// Action: select text with ID 19: go back;
	L 	19;
	T 	button_1_text;

//---------------------------------
// --- TRANSITION TO S480 ---
//---------------------------------

// Transition Logic
	SET;	// make sure RLO is high so the transition can happen when no conditions present

	A	button_1_pushed; 	// button “go back
	JCN L35;

	L   480;
	T   stepnumber;

L35: NOP 0;


//---------------------------------
// Actions (last scan)
// This is immediately executed once the stepnumber changes
//---------------------------------
	L	stepnumber;
	L	previous_stepnumber;
	<>I;
	JCN D35;

// Action: hide button_1
	CLR;
	=	button_1_visible;


D35: NOP 0;

//---------------------------------
// End of network: jump here if step not active
// Jump to end of this FB if the step has been active to avoid
// execution of another step in the same scan
//---------------------------------
	JU	ENDS;
J35: NOP 0;

//__phase_example_Step_470_END

NETWORK
TITLE = Step 480
//___phase_example_Step_480_
//================================
// test 3 buttons
//================================

// skip this network if stepnumber not equal to 480
	L 	stepnumber;
	L 	480;
	==I;
	JCN J36;

//---------------------------------
// Actions (continuouss)
//---------------------------------

// Action: show button_1
	SET;
	=	button_1_visible;

// Action: select text with ID 16: continue;
	L 	16;
	T 	button_1_text;

// Action: show button_2
	SET;
	=	button_2_visible;

// Action: select text with ID 18: cancel;
	L 	18;
	T 	button_2_text;

// Action: show button_3
	SET;
	=	button_3_visible;

// Action: select text with ID 19: go back;
	L 	19;
	T 	button_3_text;

//---------------------------------
// --- TRANSITION TO S490 ---
//---------------------------------

// Transition Logic
	SET;	// make sure RLO is high so the transition can happen when no conditions present

	A	button_1_pushed; 	// button “continue”
	A	button_2_pushed; 	// button “cancel”
	A	button_3_pushed; 	// button “go back”
	JCN L36;

	L   490;
	T   stepnumber;

L36: NOP 0;


//---------------------------------
// Actions (last scan)
// This is immediately executed once the stepnumber changes
//---------------------------------
	L	stepnumber;
	L	previous_stepnumber;
	<>I;
	JCN D36;

// Action: hide button_1
	CLR;
	=	button_1_visible;

// Action: hide button_2
	CLR;
	=	button_2_visible;

// Action: hide button_3
	CLR;
	=	button_3_visible;


D36: NOP 0;

//---------------------------------
// End of network: jump here if step not active
// Jump to end of this FB if the step has been active to avoid
// execution of another step in the same scan
//---------------------------------
	JU	ENDS;
J36: NOP 0;

//__phase_example_Step_480_END

NETWORK
TITLE = Step 490
//___phase_example_Step_490_
//================================
// test 4 buttons => not foreseen in the template, so should log an error
//================================

// skip this network if stepnumber not equal to 490
	L 	stepnumber;
	L 	490;
	==I;
	JCN J37;

//---------------------------------
// Actions (continuouss)
//---------------------------------

// Action: show button_1
	SET;
	=	button_1_visible;

// Action: select text with ID 16: continue;
	L 	16;
	T 	button_1_text;

// Action: show button_2
	SET;
	=	button_2_visible;

// Action: select text with ID 18: cancel;
	L 	18;
	T 	button_2_text;

// Action: show button_3
	SET;
	=	button_3_visible;

// Action: select text with ID 19: go back;
	L 	19;
	T 	button_3_text;

//---------------------------------
// --- TRANSITION TO S510 ---
//---------------------------------

// Transition Logic
	SET;	// make sure RLO is high so the transition can happen when no conditions present

	A	button_1_pushed; 	// button “continue”
	A	button_2_pushed; 	// button “cancel”
	A	button_3_pushed; 	// button “go back”
	JCN L37;

	L   510;
	T   stepnumber;

L37: NOP 0;


//---------------------------------
// Actions (last scan)
// This is immediately executed once the stepnumber changes
//---------------------------------
	L	stepnumber;
	L	previous_stepnumber;
	<>I;
	JCN D37;

// Action: hide button_1
	CLR;
	=	button_1_visible;

// Action: hide button_2
	CLR;
	=	button_2_visible;

// Action: hide button_3
	CLR;
	=	button_3_visible;


D37: NOP 0;

//---------------------------------
// End of network: jump here if step not active
// Jump to end of this FB if the step has been active to avoid
// execution of another step in the same scan
//---------------------------------
	JU	ENDS;
J37: NOP 0;

//__phase_example_Step_490_END

NETWORK
TITLE = Step 510
//___phase_example_Step_510_
//================================
// test message
//================================

// skip this network if stepnumber not equal to 510
	L 	stepnumber;
	L 	510;
	==I;
	JCN J38;

//---------------------------------
// Actions (continuouss)
//---------------------------------

// Action: message “add the manual ingredients”;
	L 	21;
	T 	message;

//---------------------------------
// --- TRANSITION TO S520 ---
//---------------------------------

// Transition Logic
	SET;	// make sure RLO is high so the transition can happen when no conditions present

	JCN L38;

	L   520;
	T   stepnumber;

L38: NOP 0;


//---------------------------------
// Actions (last scan)
// This is immediately executed once the stepnumber changes
//---------------------------------
	L	stepnumber;
	L	previous_stepnumber;
	<>I;
	JCN D38;

// Action: clear message;
	L 	0;
	T 	message;


D38: NOP 0;

//---------------------------------
// End of network: jump here if step not active
// Jump to end of this FB if the step has been active to avoid
// execution of another step in the same scan
//---------------------------------
	JU	ENDS;
J38: NOP 0;

//__phase_example_Step_510_END

NETWORK
TITLE = Step 520
//___phase_example_Step_520_
//================================
// test falseword with two words in transition
//================================

// skip this network if stepnumber not equal to 520
	L 	stepnumber;
	L 	520;
	==I;
	JCN J39;

//---------------------------------
// Actions (continuouss)
//---------------------------------

//---------------------------------
// --- TRANSITION TO S530 ---
//---------------------------------

// Transition Logic
	SET;	// make sure RLO is high so the transition can happen when no conditions present

	AN	XV003_OPN; 	// XV003 not opened
	JCN L39;

	L   530;
	T   stepnumber;

L39: NOP 0;


D39: NOP 0;

//---------------------------------
// End of network: jump here if step not active
// Jump to end of this FB if the step has been active to avoid
// execution of another step in the same scan
//---------------------------------
	JU	ENDS;
J39: NOP 0;

//__phase_example_Step_520_END

NETWORK
TITLE = Step 530
//___phase_example_Step_530_
//================================
// test trueword with multiple words in action
//================================

// skip this network if stepnumber not equal to 530
	L 	stepnumber;
	L 	530;
	==I;
	JCN J40;

//---------------------------------
// Actions (continuouss)
//---------------------------------

// Action: move to open position XV003
	SET;
	=	XV003_CMD;

//---------------------------------
// --- TRANSITION TO S540 ---
//---------------------------------

// Transition Logic
	SET;	// make sure RLO is high so the transition can happen when no conditions present

	JCN L40;

	L   540;
	T   stepnumber;

L40: NOP 0;


D40: NOP 0;

//---------------------------------
// End of network: jump here if step not active
// Jump to end of this FB if the step has been active to avoid
// execution of another step in the same scan
//---------------------------------
	JU	ENDS;
J40: NOP 0;

//__phase_example_Step_530_END

NETWORK
TITLE = Step 540
//___phase_example_Step_540_
//================================
// test putting controller in auto with pulseword
//================================

// skip this network if stepnumber not equal to 540
	L 	stepnumber;
	L 	540;
	==I;
	JCN J41;

//---------------------------------
// Actions (continuouss)
//---------------------------------

// Action: FIC001 auto
	SET;
	=	FIC001_AUT;

//---------------------------------
// --- TRANSITION TO S550 ---
//---------------------------------

// Transition Logic
	SET;	// make sure RLO is high so the transition can happen when no conditions present

	JCN L41;

	L   550;
	T   stepnumber;

L41: NOP 0;


D41: NOP 0;

//---------------------------------
// End of network: jump here if step not active
// Jump to end of this FB if the step has been active to avoid
// execution of another step in the same scan
//---------------------------------
	JU	ENDS;
J41: NOP 0;

//__phase_example_Step_540_END

NETWORK
TITLE = Step 550
//___phase_example_Step_550_
//================================
// test putting controller in auto with pulseword consisting of multiple words
//================================

// skip this network if stepnumber not equal to 550
	L 	stepnumber;
	L 	550;
	==I;
	JCN J42;

//---------------------------------
// Actions (continuouss)
//---------------------------------

// Action: FIC001 switch to auto
	SET;
	=	FIC001_AUT;

//---------------------------------
// --- TRANSITION TO S560 ---
//---------------------------------

// Transition Logic
	SET;	// make sure RLO is high so the transition can happen when no conditions present

	JCN L42;

	L   560;
	T   stepnumber;

L42: NOP 0;


D42: NOP 0;

//---------------------------------
// End of network: jump here if step not active
// Jump to end of this FB if the step has been active to avoid
// execution of another step in the same scan
//---------------------------------
	JU	ENDS;
J42: NOP 0;

//__phase_example_Step_550_END

NETWORK
TITLE = Step 560
//___phase_example_Step_560_
//================================
// test with pulseword in front
//================================

// skip this network if stepnumber not equal to 560
	L 	stepnumber;
	L 	560;
	==I;
	JCN J43;

//---------------------------------
// Actions (continuouss)
//---------------------------------

// Action: auto FIC001
	SET;
	=	FIC001_AUT;

//---------------------------------
// --- TRANSITION TO S570 ---
//---------------------------------

// Transition Logic
	SET;	// make sure RLO is high so the transition can happen when no conditions present

	JCN L43;

	L   570;
	T   stepnumber;

L43: NOP 0;


D43: NOP 0;

//---------------------------------
// End of network: jump here if step not active
// Jump to end of this FB if the step has been active to avoid
// execution of another step in the same scan
//---------------------------------
	JU	ENDS;
J43: NOP 0;

//__phase_example_Step_560_END

NETWORK
TITLE = Step 570
//___phase_example_Step_570_
//================================
// test with pulseword in front
//================================

// skip this network if stepnumber not equal to 570
	L 	stepnumber;
	L 	570;
	==I;
	JCN J44;

//---------------------------------
// Actions (continuouss)
//---------------------------------

// Action: switch to auto FIC001
	SET;
	=	FIC001_AUT;

//---------------------------------
// --- TRANSITION TO S580 ---
//---------------------------------

// Transition Logic
	SET;	// make sure RLO is high so the transition can happen when no conditions present

	JCN L44;

	L   580;
	T   stepnumber;

L44: NOP 0;


D44: NOP 0;

//---------------------------------
// End of network: jump here if step not active
// Jump to end of this FB if the step has been active to avoid
// execution of another step in the same scan
//---------------------------------
	JU	ENDS;
J44: NOP 0;

//__phase_example_Step_570_END

NETWORK
TITLE = Step 580
//___phase_example_Step_580_
//================================
// test steptime in s
//================================

// skip this network if stepnumber not equal to 580
	L 	stepnumber;
	L 	580;
	==I;
	JCN J45;

//---------------------------------
// Actions (continuouss)
//---------------------------------

//---------------------------------
// --- TRANSITION TO S590 ---
//---------------------------------

// Calculation:
	L 	steptime_s;
	L 	2.0;
	>R;
	=	B5;

// Transition Logic
	SET;	// make sure RLO is high so the transition can happen when no conditions present

	A	B5; 	// steptime > 2.0s
	JCN L45;

	L   590;
	T   stepnumber;

L45: NOP 0;


D45: NOP 0;

//---------------------------------
// End of network: jump here if step not active
// Jump to end of this FB if the step has been active to avoid
// execution of another step in the same scan
//---------------------------------
	JU	ENDS;
J45: NOP 0;

//__phase_example_Step_580_END

NETWORK
TITLE = Step 590
//___phase_example_Step_590_
//================================
// test steptime in m
//================================

// skip this network if stepnumber not equal to 590
	L 	stepnumber;
	L 	590;
	==I;
	JCN J46;

//---------------------------------
// Actions (continuouss)
//---------------------------------

//---------------------------------
// --- TRANSITION TO S600 ---
//---------------------------------

// Calculation:
	L 	steptime_m;
	L 	1.50;
	>R;
	=	B6;

// Transition Logic
	SET;	// make sure RLO is high so the transition can happen when no conditions present

	A	B6; 	// steptime > 1.50m
	JCN L46;

	L   600;
	T   stepnumber;

L46: NOP 0;


D46: NOP 0;

//---------------------------------
// End of network: jump here if step not active
// Jump to end of this FB if the step has been active to avoid
// execution of another step in the same scan
//---------------------------------
	JU	ENDS;
J46: NOP 0;

//__phase_example_Step_590_END

NETWORK
TITLE = Step 600
//___phase_example_Step_600_
//================================
// test steptime in h
//================================

// skip this network if stepnumber not equal to 600
	L 	stepnumber;
	L 	600;
	==I;
	JCN J47;

//---------------------------------
// Actions (continuouss)
//---------------------------------

//---------------------------------
// --- TRANSITION TO S610 ---
//---------------------------------

// Calculation:
	L 	steptime_h;
	L 	4.3;
	>R;
	=	B7;

// Transition Logic
	SET;	// make sure RLO is high so the transition can happen when no conditions present

	A	B7; 	// steptime > 4.3h
	JCN L47;

	L   610;
	T   stepnumber;

L47: NOP 0;


D47: NOP 0;

//---------------------------------
// End of network: jump here if step not active
// Jump to end of this FB if the step has been active to avoid
// execution of another step in the same scan
//---------------------------------
	JU	ENDS;
J47: NOP 0;

//__phase_example_Step_600_END

NETWORK
TITLE = Step 610
//___phase_example_Step_610_
//================================
// test steptime with unit separated by space => still works (because it takes the last character)
//================================

// skip this network if stepnumber not equal to 610
	L 	stepnumber;
	L 	610;
	==I;
	JCN J48;

//---------------------------------
// Actions (continuouss)
//---------------------------------

//---------------------------------
// --- TRANSITION TO S640 ---
//---------------------------------

// Calculation:
	L 	steptime_m;
	L 	1.50;
	>R;
	=	B8;

// Transition Logic
	SET;	// make sure RLO is high so the transition can happen when no conditions present

	A	B8; 	// steptime > 1.50 m
	JCN L48;

	L   640;
	T   stepnumber;

L48: NOP 0;


D48: NOP 0;

//---------------------------------
// End of network: jump here if step not active
// Jump to end of this FB if the step has been active to avoid
// execution of another step in the same scan
//---------------------------------
	JU	ENDS;
J48: NOP 0;

//__phase_example_Step_610_END

NETWORK
TITLE = Step 640
//___phase_example_Step_640_
//================================
// test steptime with variable with unit
//================================

// skip this network if stepnumber not equal to 640
	L 	stepnumber;
	L 	640;
	==I;
	JCN J49;

//---------------------------------
// Actions (continuouss)
//---------------------------------

//---------------------------------
// --- TRANSITION TO S650 ---
//---------------------------------

// Calculation:
	L 	steptime_h;
	L 	timesetting;
	>R;
	=	B9;

// Transition Logic
	SET;	// make sure RLO is high so the transition can happen when no conditions present

	A	B9; 	// steptime > timesetting
	JCN L49;

	L   650;
	T   stepnumber;

L49: NOP 0;


D49: NOP 0;

//---------------------------------
// End of network: jump here if step not active
// Jump to end of this FB if the step has been active to avoid
// execution of another step in the same scan
//---------------------------------
	JU	ENDS;
J49: NOP 0;

//__phase_example_Step_640_END

NETWORK
TITLE = Step 650
//___phase_example_Step_650_
//================================
// reset a timer
//================================

// skip this network if stepnumber not equal to 650
	L 	stepnumber;
	L 	650;
	==I;
	JCN J50;

//---------------------------------
// Actions (continuouss)
//---------------------------------

// Action: reset timer_dosing;
	L 	0.0;
	T 	timer_dosing_s;

//---------------------------------
// --- TRANSITION TO S660 ---
//---------------------------------

// Transition Logic
	SET;	// make sure RLO is high so the transition can happen when no conditions present

	JCN L50;

	L   660;
	T   stepnumber;

L50: NOP 0;


D50: NOP 0;

//---------------------------------
// End of network: jump here if step not active
// Jump to end of this FB if the step has been active to avoid
// execution of another step in the same scan
//---------------------------------
	JU	ENDS;
J50: NOP 0;

//__phase_example_Step_650_END

NETWORK
TITLE = Step 660
//___phase_example_Step_660_
//================================
// start a timer
//================================

// skip this network if stepnumber not equal to 660
	L 	stepnumber;
	L 	660;
	==I;
	JCN J51;

//---------------------------------
// Actions (continuouss)
//---------------------------------

// Action: start timer_mixing
	CLR;
	=	timer_mixing_pause;

//---------------------------------
// --- TRANSITION TO S670 ---
//---------------------------------

// Transition Logic
	SET;	// make sure RLO is high so the transition can happen when no conditions present

	JCN L51;

	L   670;
	T   stepnumber;

L51: NOP 0;


D51: NOP 0;

//---------------------------------
// End of network: jump here if step not active
// Jump to end of this FB if the step has been active to avoid
// execution of another step in the same scan
//---------------------------------
	JU	ENDS;
J51: NOP 0;

//__phase_example_Step_660_END

NETWORK
TITLE = Step 670
//___phase_example_Step_670_
//================================
// pause a timer
//================================

// skip this network if stepnumber not equal to 670
	L 	stepnumber;
	L 	670;
	==I;
	JCN J52;

//---------------------------------
// Actions (continuouss)
//---------------------------------

// Action: pause timer_circulation
	SET;
	=	timer_circulation_pause;

//---------------------------------
// --- TRANSITION TO S680 ---
//---------------------------------

// Transition Logic
	SET;	// make sure RLO is high so the transition can happen when no conditions present

	JCN L52;

	L   680;
	T   stepnumber;

L52: NOP 0;


D52: NOP 0;

//---------------------------------
// End of network: jump here if step not active
// Jump to end of this FB if the step has been active to avoid
// execution of another step in the same scan
//---------------------------------
	JU	ENDS;
J52: NOP 0;

//__phase_example_Step_670_END

NETWORK
TITLE = Step 680
//___phase_example_Step_680_
//================================
// test timer in m
//================================

// skip this network if stepnumber not equal to 680
	L 	stepnumber;
	L 	680;
	==I;
	JCN J53;

//---------------------------------
// Actions (continuouss)
//---------------------------------

//---------------------------------
// --- TRANSITION TO S690 ---
//---------------------------------

// Calculation:
	L 	timer_dosing_m;
	L 	5.2;
	>=R;
	=	B10;

// Transition Logic
	SET;	// make sure RLO is high so the transition can happen when no conditions present

	A	B10; 	// timer_dosing >= 5.2 m
	JCN L53;

	L   690;
	T   stepnumber;

L53: NOP 0;


D53: NOP 0;

//---------------------------------
// End of network: jump here if step not active
// Jump to end of this FB if the step has been active to avoid
// execution of another step in the same scan
//---------------------------------
	JU	ENDS;
J53: NOP 0;

//__phase_example_Step_680_END

NETWORK
TITLE = Step 690
//___phase_example_Step_690_
//================================
// test timer with variable with unit
//================================

// skip this network if stepnumber not equal to 690
	L 	stepnumber;
	L 	690;
	==I;
	JCN J54;

//---------------------------------
// Actions (continuouss)
//---------------------------------

//---------------------------------
// --- TRANSITION TO S700 ---
//---------------------------------

// Calculation:
	L 	timer_circulation_h;
	L 	timesetting;
	<R;
	=	B11;

// Transition Logic
	SET;	// make sure RLO is high so the transition can happen when no conditions present

	A	B11; 	// timer_circulation < timesetting
	JCN L54;

	L   700;
	T   stepnumber;

L54: NOP 0;


D54: NOP 0;

//---------------------------------
// End of network: jump here if step not active
// Jump to end of this FB if the step has been active to avoid
// execution of another step in the same scan
//---------------------------------
	JU	ENDS;
J54: NOP 0;

//__phase_example_Step_690_END

NETWORK
TITLE = Step 700
//___phase_example_Step_700_
//================================
// test putting a controller in manual
//================================

// skip this network if stepnumber not equal to 700
	L 	stepnumber;
	L 	700;
	==I;
	JCN J55;

//---------------------------------
// Actions (continuouss)
//---------------------------------

// Action: FIC001 manual
	CLR;
	=	FIC001_AUT;

//---------------------------------
// --- TRANSITION TO S710 ---
//---------------------------------

// Transition Logic
	SET;	// make sure RLO is high so the transition can happen when no conditions present

	JCN L55;

	L   710;
	T   stepnumber;

L55: NOP 0;


D55: NOP 0;

//---------------------------------
// End of network: jump here if step not active
// Jump to end of this FB if the step has been active to avoid
// execution of another step in the same scan
//---------------------------------
	JU	ENDS;
J55: NOP 0;

//__phase_example_Step_700_END

NETWORK
TITLE = Step 710
//___phase_example_Step_710_
//================================
// test putting a controller in manual while changing the output value
//================================

// skip this network if stepnumber not equal to 710
	L 	stepnumber;
	L 	710;
	==I;
	JCN J56;

//---------------------------------
// Actions (first scan)
//---------------------------------
	A	initial_scan;
	JCN   C56;

// Action: FIC001_VAL_OUT = 20.0;
	L 	20.0;
	T 	FIC001_VAL_OUT;

// Action: FIC001_SET_OUT = true
	SET;
	=	FIC001_SET_OUT;

	JU	D56;	//skip the continuous steps and transition during the initial scan
C56: NOP   0;


//---------------------------------
// Actions (continuouss)
//---------------------------------

// Action: FIC001 manual 20.0
	CLR;
	=	FIC001_AUT;

// Action: FIC001_SET_OUT = false
	CLR;
	=	FIC001_SET_OUT;

//---------------------------------
// --- TRANSITION TO S720 ---
//---------------------------------

// Transition Logic
	SET;	// make sure RLO is high so the transition can happen when no conditions present

	JCN L56;

	L   720;
	T   stepnumber;

L56: NOP 0;


D56: NOP 0;

//---------------------------------
// End of network: jump here if step not active
// Jump to end of this FB if the step has been active to avoid
// execution of another step in the same scan
//---------------------------------
	JU	ENDS;
J56: NOP 0;

//__phase_example_Step_710_END

NETWORK
TITLE = Step 720
//___phase_example_Step_720_
//================================
// test putting a controller in manual while changing the output value that has a unit
//================================

// skip this network if stepnumber not equal to 720
	L 	stepnumber;
	L 	720;
	==I;
	JCN J57;

//---------------------------------
// Actions (first scan)
//---------------------------------
	A	initial_scan;
	JCN   C57;

// Action: FIC001_VAL_OUT = 20.0;
	L 	20.0;
	T 	FIC001_VAL_OUT;

// Action: FIC001_SET_OUT = true
	SET;
	=	FIC001_SET_OUT;

	JU	D57;	//skip the continuous steps and transition during the initial scan
C57: NOP   0;


//---------------------------------
// Actions (continuouss)
//---------------------------------

// Action: FIC001 manual 20.0 Hz
	CLR;
	=	FIC001_AUT;

// Action: FIC001_SET_OUT = false
	CLR;
	=	FIC001_SET_OUT;

//---------------------------------
// --- TRANSITION TO S730 ---
//---------------------------------

// Transition Logic
	SET;	// make sure RLO is high so the transition can happen when no conditions present

	JCN L57;

	L   730;
	T   stepnumber;

L57: NOP 0;


D57: NOP 0;

//---------------------------------
// End of network: jump here if step not active
// Jump to end of this FB if the step has been active to avoid
// execution of another step in the same scan
//---------------------------------
	JU	ENDS;
J57: NOP 0;

//__phase_example_Step_720_END

NETWORK
TITLE = Step 730
//___phase_example_Step_730_
//================================
// without space
//================================

// skip this network if stepnumber not equal to 730
	L 	stepnumber;
	L 	730;
	==I;
	JCN J58;

//---------------------------------
// Actions (first scan)
//---------------------------------
	A	initial_scan;
	JCN   C58;

// Action: FIC001_VAL_OUT = 20.0;
	L 	20.0;
	T 	FIC001_VAL_OUT;

// Action: FIC001_SET_OUT = true
	SET;
	=	FIC001_SET_OUT;

	JU	D58;	//skip the continuous steps and transition during the initial scan
C58: NOP   0;


//---------------------------------
// Actions (continuouss)
//---------------------------------

// Action: FIC001 manual 20.0Hz
	CLR;
	=	FIC001_AUT;

// Action: FIC001_SET_OUT = false
	CLR;
	=	FIC001_SET_OUT;

//---------------------------------
// --- TRANSITION TO S740 ---
//---------------------------------

// Transition Logic
	SET;	// make sure RLO is high so the transition can happen when no conditions present

	JCN L58;

	L   740;
	T   stepnumber;

L58: NOP 0;


D58: NOP 0;

//---------------------------------
// End of network: jump here if step not active
// Jump to end of this FB if the step has been active to avoid
// execution of another step in the same scan
//---------------------------------
	JU	ENDS;
J58: NOP 0;

//__phase_example_Step_730_END

NETWORK
TITLE = Step 740
//___phase_example_Step_740_
//================================
// put PID controller in auto
//================================

// skip this network if stepnumber not equal to 740
	L 	stepnumber;
	L 	740;
	==I;
	JCN J59;

//---------------------------------
// Actions (continuouss)
//---------------------------------

// Action: FIC001 auto
	SET;
	=	FIC001_AUT;

//---------------------------------
// --- TRANSITION TO S750 ---
//---------------------------------

// Transition Logic
	SET;	// make sure RLO is high so the transition can happen when no conditions present

	JCN L59;

	L   750;
	T   stepnumber;

L59: NOP 0;


D59: NOP 0;

//---------------------------------
// End of network: jump here if step not active
// Jump to end of this FB if the step has been active to avoid
// execution of another step in the same scan
//---------------------------------
	JU	ENDS;
J59: NOP 0;

//__phase_example_Step_740_END

NETWORK
TITLE = Step 750
//___phase_example_Step_750_
//================================
// auto with setpoint
//================================

// skip this network if stepnumber not equal to 750
	L 	stepnumber;
	L 	750;
	==I;
	JCN J60;

//---------------------------------
// Actions (first scan)
//---------------------------------
	A	initial_scan;
	JCN   C60;

// Action: FIC001_SP = 80.0;
	L 	80.0;
	T 	FIC001_SP;

// Action: FIC001_SET_SP = true
	SET;
	=	FIC001_SET_SP;

	JU	D60;	//skip the continuous steps and transition during the initial scan
C60: NOP   0;


//---------------------------------
// Actions (continuouss)
//---------------------------------

// Action: FIC001 auto 80.0%
	SET;
	=	FIC001_AUT;

// Action: FIC001_SET_SP = false
	CLR;
	=	FIC001_SET_SP;

//---------------------------------
// --- TRANSITION TO S760 ---
//---------------------------------

// Transition Logic
	SET;	// make sure RLO is high so the transition can happen when no conditions present

	JCN L60;

	L   760;
	T   stepnumber;

L60: NOP 0;


D60: NOP 0;

//---------------------------------
// End of network: jump here if step not active
// Jump to end of this FB if the step has been active to avoid
// execution of another step in the same scan
//---------------------------------
	JU	ENDS;
J60: NOP 0;

//__phase_example_Step_750_END

NETWORK
TITLE = Step 760
//___phase_example_Step_760_
//================================
// internal mode
//================================

// skip this network if stepnumber not equal to 760
	L 	stepnumber;
	L 	760;
	==I;
	JCN J61;

//---------------------------------
// Actions (continuouss)
//---------------------------------

// Action: FIC001 internal
	CLR;
	=	FIC001_EXT;

//---------------------------------
// --- TRANSITION TO S770 ---
//---------------------------------

// Transition Logic
	SET;	// make sure RLO is high so the transition can happen when no conditions present

	JCN L61;

	L   770;
	T   stepnumber;

L61: NOP 0;


D61: NOP 0;

//---------------------------------
// End of network: jump here if step not active
// Jump to end of this FB if the step has been active to avoid
// execution of another step in the same scan
//---------------------------------
	JU	ENDS;
J61: NOP 0;

//__phase_example_Step_760_END

NETWORK
TITLE = Step 770
//___phase_example_Step_770_
//================================
// internal mode with value
//================================

// skip this network if stepnumber not equal to 770
	L 	stepnumber;
	L 	770;
	==I;
	JCN J62;

//---------------------------------
// Actions (first scan)
//---------------------------------
	A	initial_scan;
	JCN   C62;

// Action: FIC001_SP = 80.0;
	L 	80.0;
	T 	FIC001_SP;

// Action: FIC001_SET_SP = true
	SET;
	=	FIC001_SET_SP;

	JU	D62;	//skip the continuous steps and transition during the initial scan
C62: NOP   0;


//---------------------------------
// Actions (continuouss)
//---------------------------------

// Action: FIC001 internal 80.0
	CLR;
	=	FIC001_EXT;

// Action: FIC001_SET_SP = false
	CLR;
	=	FIC001_SET_SP;

//---------------------------------
// --- TRANSITION TO S780 ---
//---------------------------------

// Transition Logic
	SET;	// make sure RLO is high so the transition can happen when no conditions present

	JCN L62;

	L   780;
	T   stepnumber;

L62: NOP 0;


D62: NOP 0;

//---------------------------------
// End of network: jump here if step not active
// Jump to end of this FB if the step has been active to avoid
// execution of another step in the same scan
//---------------------------------
	JU	ENDS;
J62: NOP 0;

//__phase_example_Step_770_END

NETWORK
TITLE = Step 780
//___phase_example_Step_780_
//================================
// value with unit
//================================

// skip this network if stepnumber not equal to 780
	L 	stepnumber;
	L 	780;
	==I;
	JCN J63;

//---------------------------------
// Actions (first scan)
//---------------------------------
	A	initial_scan;
	JCN   C63;

// Action: FIC001_SP = 80.0;
	L 	80.0;
	T 	FIC001_SP;

// Action: FIC001_SET_SP = true
	SET;
	=	FIC001_SET_SP;

	JU	D63;	//skip the continuous steps and transition during the initial scan
C63: NOP   0;


//---------------------------------
// Actions (continuouss)
//---------------------------------

// Action: FIC001 internal 80.0 %
	CLR;
	=	FIC001_EXT;

// Action: FIC001_SET_SP = false
	CLR;
	=	FIC001_SET_SP;

//---------------------------------
// --- TRANSITION TO S790 ---
//---------------------------------

// Transition Logic
	SET;	// make sure RLO is high so the transition can happen when no conditions present

	JCN L63;

	L   790;
	T   stepnumber;

L63: NOP 0;


D63: NOP 0;

//---------------------------------
// End of network: jump here if step not active
// Jump to end of this FB if the step has been active to avoid
// execution of another step in the same scan
//---------------------------------
	JU	ENDS;
J63: NOP 0;

//__phase_example_Step_780_END

NETWORK
TITLE = Step 790
//___phase_example_Step_790_
//================================
// without space
//================================

// skip this network if stepnumber not equal to 790
	L 	stepnumber;
	L 	790;
	==I;
	JCN J64;

//---------------------------------
// Actions (first scan)
//---------------------------------
	A	initial_scan;
	JCN   C64;

// Action: FIC001_SP = 80.0;
	L 	80.0;
	T 	FIC001_SP;

// Action: FIC001_SET_SP = true
	SET;
	=	FIC001_SET_SP;

	JU	D64;	//skip the continuous steps and transition during the initial scan
C64: NOP   0;


//---------------------------------
// Actions (continuouss)
//---------------------------------

// Action: FIC001 internal80.0%
	CLR;
	=	FIC001_EXT;

// Action: FIC001_SET_SP = false
	CLR;
	=	FIC001_SET_SP;

//---------------------------------
// --- TRANSITION TO S810 ---
//---------------------------------

// Transition Logic
	SET;	// make sure RLO is high so the transition can happen when no conditions present

	JCN L64;

	L   810;
	T   stepnumber;

L64: NOP 0;


D64: NOP 0;

//---------------------------------
// End of network: jump here if step not active
// Jump to end of this FB if the step has been active to avoid
// execution of another step in the same scan
//---------------------------------
	JU	ENDS;
J64: NOP 0;

//__phase_example_Step_790_END

NETWORK
TITLE = Step 810
//___phase_example_Step_810_
//================================
// external mode
//================================

// skip this network if stepnumber not equal to 810
	L 	stepnumber;
	L 	810;
	==I;
	JCN J65;

//---------------------------------
// Actions (continuouss)
//---------------------------------

// Action: FIC001 external
	SET;
	=	FIC001_EXT;

//---------------------------------
// --- TRANSITION TO S820 ---
//---------------------------------

// Transition Logic
	SET;	// make sure RLO is high so the transition can happen when no conditions present

	JCN L65;

	L   820;
	T   stepnumber;

L65: NOP 0;


D65: NOP 0;

//---------------------------------
// End of network: jump here if step not active
// Jump to end of this FB if the step has been active to avoid
// execution of another step in the same scan
//---------------------------------
	JU	ENDS;
J65: NOP 0;

//__phase_example_Step_810_END

NETWORK
TITLE = Step 820
//___phase_example_Step_820_
//================================
// test direct access to a CM instance in dot-format in the assignment => should convert to suffix
//================================

// skip this network if stepnumber not equal to 820
	L 	stepnumber;
	L 	820;
	==I;
	JCN J66;

//---------------------------------
// Actions (continuouss)
//---------------------------------

// Action: XV008.AUT_OP = true
	SET;
	=	XV008_CMD;

//---------------------------------
// --- TRANSITION TO S830 ---
//---------------------------------

// Transition Logic
	SET;	// make sure RLO is high so the transition can happen when no conditions present

	JCN L66;

	L   830;
	T   stepnumber;

L66: NOP 0;


D66: NOP 0;

//---------------------------------
// End of network: jump here if step not active
// Jump to end of this FB if the step has been active to avoid
// execution of another step in the same scan
//---------------------------------
	JU	ENDS;
J66: NOP 0;

//__phase_example_Step_820_END

NETWORK
TITLE = Step 830
//___phase_example_Step_830_
//================================
// test direct access to a CM in dot-notation in the evaluation => should convert to suffix
//================================

// skip this network if stepnumber not equal to 830
	L 	stepnumber;
	L 	830;
	==I;
	JCN J67;

//---------------------------------
// Actions (continuouss)
//---------------------------------

//---------------------------------
// --- TRANSITION TO S840 ---
//---------------------------------

// Transition Logic
	SET;	// make sure RLO is high so the transition can happen when no conditions present

	A	XV008_OPN; 	// XV008.QOPEN = true
	JCN L67;

	L   840;
	T   stepnumber;

L67: NOP 0;


D67: NOP 0;

//---------------------------------
// End of network: jump here if step not active
// Jump to end of this FB if the step has been active to avoid
// execution of another step in the same scan
//---------------------------------
	JU	ENDS;
J67: NOP 0;

//__phase_example_Step_830_END

NETWORK
TITLE = Step 840
//___phase_example_Step_840_
//================================
// test dot-format to Linked CM in assignment => should convert to suffix
//================================

// skip this network if stepnumber not equal to 840
	L 	stepnumber;
	L 	840;
	==I;
	JCN J68;

//---------------------------------
// Actions (continuouss)
//---------------------------------

// Action: XV003.AUT_OP = true
	SET;
	=	XV003_CMD;

//---------------------------------
// --- TRANSITION TO S850 ---
//---------------------------------

// Transition Logic
	SET;	// make sure RLO is high so the transition can happen when no conditions present

	JCN L68;

	L   850;
	T   stepnumber;

L68: NOP 0;


D68: NOP 0;

//---------------------------------
// End of network: jump here if step not active
// Jump to end of this FB if the step has been active to avoid
// execution of another step in the same scan
//---------------------------------
	JU	ENDS;
J68: NOP 0;

//__phase_example_Step_840_END

NETWORK
TITLE = Step 850
//___phase_example_Step_850_
//================================
// test dot-format from Linked CM in evaluation =>should convert to suffix
//================================

// skip this network if stepnumber not equal to 850
	L 	stepnumber;
	L 	850;
	==I;
	JCN J69;

//---------------------------------
// Actions (continuouss)
//---------------------------------

//---------------------------------
// --- TRANSITION TO S860 ---
//---------------------------------

// Transition Logic
	SET;	// make sure RLO is high so the transition can happen when no conditions present

	A	XV003_OPN; 	// XV003.QOPEN = true
	JCN L69;

	L   860;
	T   stepnumber;

L69: NOP 0;


D69: NOP 0;

//---------------------------------
// End of network: jump here if step not active
// Jump to end of this FB if the step has been active to avoid
// execution of another step in the same scan
//---------------------------------
	JU	ENDS;
J69: NOP 0;

//__phase_example_Step_850_END

NETWORK
TITLE = Step 860
//___phase_example_Step_860_
//================================
// test direct access to an EM instance in dot-format in the assignment => should stay in dot-format
//================================

// skip this network if stepnumber not equal to 860
	L 	stepnumber;
	L 	860;
	==I;
	JCN J70;

//---------------------------------
// Actions (continuouss)
//---------------------------------

// Action: EM_Instance_4.Pressure_SP  = 4.2;
	L 	4.2;
	T 	%%prefix_EM_instances%%EM_Instance_4.Pressure_SP;

//---------------------------------
// --- TRANSITION TO S870 ---
//---------------------------------

// Transition Logic
	SET;	// make sure RLO is high so the transition can happen when no conditions present

	JCN L70;

	L   870;
	T   stepnumber;

L70: NOP 0;


D70: NOP 0;

//---------------------------------
// End of network: jump here if step not active
// Jump to end of this FB if the step has been active to avoid
// execution of another step in the same scan
//---------------------------------
	JU	ENDS;
J70: NOP 0;

//__phase_example_Step_860_END

NETWORK
TITLE = Step 870
//___phase_example_Step_870_
//================================
// test direct access to a EM in dot-notation in the evaluation => should stay in dot-format
//================================

// skip this network if stepnumber not equal to 870
	L 	stepnumber;
	L 	870;
	==I;
	JCN J71;

//---------------------------------
// Actions (continuouss)
//---------------------------------

//---------------------------------
// --- TRANSITION TO S880 ---
//---------------------------------

// Calculation: %%prefix_EM_instances%%EM_Instance_4.Level >= 50.0
	L 	%%prefix_EM_instances%%EM_Instance_4.Level;
	L 	50.0;
	>=R;
	=	B12;

// Transition Logic
	SET;	// make sure RLO is high so the transition can happen when no conditions present

	A	B12; 	// EM_Instance_4.Level >= 50.0
	JCN L71;

	L   880;
	T   stepnumber;

L71: NOP 0;


D71: NOP 0;

//---------------------------------
// End of network: jump here if step not active
// Jump to end of this FB if the step has been active to avoid
// execution of another step in the same scan
//---------------------------------
	JU	ENDS;
J71: NOP 0;

//__phase_example_Step_870_END

NETWORK
TITLE = Step 880
//___phase_example_Step_880_
//================================
// test dot-format to Linked EM in assignment => should stay in dot-format
//================================

// skip this network if stepnumber not equal to 880
	L 	stepnumber;
	L 	880;
	==I;
	JCN J72;

//---------------------------------
// Actions (continuouss)
//---------------------------------

// Action: Some_Dyn_EM.Pressure_SP  = 4.2;
	L 	4.2;
	T 	Some_Dyn_EM.Pressure_SP;

//---------------------------------
// --- TRANSITION TO S890 ---
//---------------------------------

// Transition Logic
	SET;	// make sure RLO is high so the transition can happen when no conditions present

	JCN L72;

	L   890;
	T   stepnumber;

L72: NOP 0;


D72: NOP 0;

//---------------------------------
// End of network: jump here if step not active
// Jump to end of this FB if the step has been active to avoid
// execution of another step in the same scan
//---------------------------------
	JU	ENDS;
J72: NOP 0;

//__phase_example_Step_880_END

NETWORK
TITLE = Step 890
//___phase_example_Step_890_
//================================
// test dot-format from Linked EM in evaluation =>should stay in dot-format
//================================

// skip this network if stepnumber not equal to 890
	L 	stepnumber;
	L 	890;
	==I;
	JCN J73;

//---------------------------------
// Actions (continuouss)
//---------------------------------

//---------------------------------
// --- TRANSITION TO S910 ---
//---------------------------------

// Calculation: Some_Dyn_EM.Level >= 50.0
	L 	Some_Dyn_EM.Level;
	L 	50.0;
	>=R;
	=	B13;

// Transition Logic
	SET;	// make sure RLO is high so the transition can happen when no conditions present

	A	B13; 	// Some_Dyn_EM.Level >= 50.0
	JCN L73;

	L   910;
	T   stepnumber;

L73: NOP 0;


D73: NOP 0;

//---------------------------------
// End of network: jump here if step not active
// Jump to end of this FB if the step has been active to avoid
// execution of another step in the same scan
//---------------------------------
	JU	ENDS;
J73: NOP 0;

//__phase_example_Step_890_END

NETWORK
TITLE = Step 910
//___phase_example_Step_910_
//================================
// test suffix-format to Linked EM in assignment => should convert to dot-format
// Some_Dyn_EM_P_SP  = 4.3
// Not longer supported: only support dot notation because it is more natural to use. Keep it simple.
//================================

// skip this network if stepnumber not equal to 910
	L 	stepnumber;
	L 	910;
	==I;
	JCN J74;

//---------------------------------
// Actions (continuouss)
//---------------------------------

//---------------------------------
// --- TRANSITION TO S920 ---
//---------------------------------

// Transition Logic
	SET;	// make sure RLO is high so the transition can happen when no conditions present

	JCN L74;

	L   920;
	T   stepnumber;

L74: NOP 0;


D74: NOP 0;

//---------------------------------
// End of network: jump here if step not active
// Jump to end of this FB if the step has been active to avoid
// execution of another step in the same scan
//---------------------------------
	JU	ENDS;
J74: NOP 0;

//__phase_example_Step_910_END

NETWORK
TITLE = Step 920
//___phase_example_Step_920_
//================================
// test suffix-format from Linked EM in evaluation =>should convert to dot-format
// Cancelled support for this: simplify and only allow dot format
//================================

// skip this network if stepnumber not equal to 920
	L 	stepnumber;
	L 	920;
	==I;
	JCN J75;

//---------------------------------
// Actions (continuouss)
//---------------------------------

//---------------------------------
// --- TRANSITION TO S930 ---
//---------------------------------

// Transition Logic
	SET;	// make sure RLO is high so the transition can happen when no conditions present

	JCN L75;

	L   930;
	T   stepnumber;

L75: NOP 0;


D75: NOP 0;

//---------------------------------
// End of network: jump here if step not active
// Jump to end of this FB if the step has been active to avoid
// execution of another step in the same scan
//---------------------------------
	JU	ENDS;
J75: NOP 0;

//__phase_example_Step_920_END

NETWORK
TITLE = Step 930
//___phase_example_Step_930_
//================================
// write a bool
//================================

// skip this network if stepnumber not equal to 930
	L 	stepnumber;
	L 	930;
	==I;
	JCN J76;

//---------------------------------
// Actions (continuouss)
//---------------------------------

// Action: some_bool_out = true
	SET;
	=	some_bool_out;

//---------------------------------
// --- TRANSITION TO S940 ---
//---------------------------------

// Transition Logic
	SET;	// make sure RLO is high so the transition can happen when no conditions present

	JCN L76;

	L   940;
	T   stepnumber;

L76: NOP 0;


D76: NOP 0;

//---------------------------------
// End of network: jump here if step not active
// Jump to end of this FB if the step has been active to avoid
// execution of another step in the same scan
//---------------------------------
	JU	ENDS;
J76: NOP 0;

//__phase_example_Step_930_END

NETWORK
TITLE = Step 940
//___phase_example_Step_940_
//================================
// test absolute value calculation
//================================

// skip this network if stepnumber not equal to 940
	L 	stepnumber;
	L 	940;
	==I;
	JCN J77;

//---------------------------------
// Actions (continuouss)
//---------------------------------

// Action: test1 = abs(2.3);
	L	2.3;
	ABS;
	T	test1;

// Action: test2 = abs(test1);
	L	test1;
	ABS;
	T	test2;

//---------------------------------
// --- TRANSITION TO S950 ---
//---------------------------------

// Transition Logic
	SET;	// make sure RLO is high so the transition can happen when no conditions present

	JCN L77;

	L   950;
	T   stepnumber;

L77: NOP 0;


D77: NOP 0;

//---------------------------------
// End of network: jump here if step not active
// Jump to end of this FB if the step has been active to avoid
// execution of another step in the same scan
//---------------------------------
	JU	ENDS;
J77: NOP 0;

//__phase_example_Step_940_END

NETWORK
TITLE = Step 950
//___phase_example_Step_950_
//================================
// test absolute value calculation to int value
//================================

// skip this network if stepnumber not equal to 950
	L 	stepnumber;
	L 	950;
	==I;
	JCN J78;

//---------------------------------
// Actions (continuouss)
//---------------------------------

// Action: intvar = abs(4.6);
	L	4.6;
	ABS;
	RND;
	T	intvar;

// Action: intvar = abs(test1);
	L	test1;
	ABS;
	RND;
	T	intvar;

// Calculation: abs(3.2)
	L 	3.2;
	ABS;
	T 	V16;

// Calculation: intvar + (abs(3.2))
	L 	intvar;
	ITD;
DTR;
	L 	V16;
	+R;
	T 	V17;

// Action: intvar = intvar + (intvar+ abs(3.2));
	L	intvar;
	ITD;
DTR;
	L	V17;
	+I;
	RND;
	T	intvar;

//---------------------------------
// --- TRANSITION TO S960 ---
//---------------------------------

// Transition Logic
	SET;	// make sure RLO is high so the transition can happen when no conditions present

	JCN L78;

	L   960;
	T   stepnumber;

L78: NOP 0;


D78: NOP 0;

//---------------------------------
// End of network: jump here if step not active
// Jump to end of this FB if the step has been active to avoid
// execution of another step in the same scan
//---------------------------------
	JU	ENDS;
J78: NOP 0;

//__phase_example_Step_950_END

NETWORK
TITLE = Step 960
//___phase_example_Step_960_
//================================
// test absolut function of another calc
//================================

// skip this network if stepnumber not equal to 960
	L 	stepnumber;
	L 	960;
	==I;
	JCN J79;

//---------------------------------
// Actions (continuouss)
//---------------------------------

// Calculation: test1 + test2
	L 	test1;
	L 	test2;
	+R;
	T 	V18;

// Action: test1 = abs(test1 + test2);
	L	V18;
	ABS;
	T	test1;

//---------------------------------
// --- TRANSITION TO S970 ---
//---------------------------------

// Transition Logic
	SET;	// make sure RLO is high so the transition can happen when no conditions present

	JCN L79;

	L   970;
	T   stepnumber;

L79: NOP 0;


D79: NOP 0;

//---------------------------------
// End of network: jump here if step not active
// Jump to end of this FB if the step has been active to avoid
// execution of another step in the same scan
//---------------------------------
	JU	ENDS;
J79: NOP 0;

//__phase_example_Step_960_END

NETWORK
TITLE = Step 970
//___phase_example_Step_970_
//================================
// test multiple transitions in one step
//================================

// skip this network if stepnumber not equal to 970
	L 	stepnumber;
	L 	970;
	==I;
	JCN J80;

//---------------------------------
// Actions (continuouss)
//---------------------------------

//---------------------------------
// --- TRANSITION TO S980 ---
//---------------------------------

// Calculation: foo > 1.0
	L 	foo;
	L 	1.0;
	>R;
	=	B14;

// Transition Logic
	SET;	// make sure RLO is high so the transition can happen when no conditions present

	A	B14; 	// foo > 1.0
	JCN L80;

	L   980;
	T   stepnumber;

L80: NOP 0;

//---------------------------------
// --- TRANSITION TO S990 ---
//---------------------------------

// Calculation: foo <= 1.0
	L 	foo;
	L 	1.0;
	<=R;
	=	B15;

// Transition Logic
	SET;	// make sure RLO is high so the transition can happen when no conditions present

	A	B15; 	// foo <= 1.0
	JCN L81;

	L   990;
	T   stepnumber;

L81: NOP 0;


D80: NOP 0;

//---------------------------------
// End of network: jump here if step not active
// Jump to end of this FB if the step has been active to avoid
// execution of another step in the same scan
//---------------------------------
	JU	ENDS;
J80: NOP 0;

//__phase_example_Step_970_END

NETWORK
TITLE = Step 980
//___phase_example_Step_980_
//================================
// assignment where the right part is a boolean variable
//================================

// skip this network if stepnumber not equal to 980
	L 	stepnumber;
	L 	980;
	==I;
	JCN J81;

//---------------------------------
// Actions (continuouss)
//---------------------------------

// Action: Bool1 = Bool2
	A	Bool2;
	=	Bool1;

//---------------------------------
// --- TRANSITION TO S990 ---
//---------------------------------

// Transition Logic
	SET;	// make sure RLO is high so the transition can happen when no conditions present

	JCN L82;

	L   990;
	T   stepnumber;

L82: NOP 0;


D81: NOP 0;

//---------------------------------
// End of network: jump here if step not active
// Jump to end of this FB if the step has been active to avoid
// execution of another step in the same scan
//---------------------------------
	JU	ENDS;
J81: NOP 0;

//__phase_example_Step_980_END

NETWORK
TITLE = Step 990
//___phase_example_Step_990_
//================================
// comparison where the right part is a boolen variable
//================================

// skip this network if stepnumber not equal to 990
	L 	stepnumber;
	L 	990;
	==I;
	JCN J82;

//---------------------------------
// Actions (continuouss)
//---------------------------------

//---------------------------------
// --- TRANSITION TO S1000 ---
//---------------------------------

// Calculation: Bool1 == Bool2
	X 	Bool1;
	X 	Bool2;
	NOT;
	=	B16;	// use of XOR to compare two bools

// Transition Logic
	SET;	// make sure RLO is high so the transition can happen when no conditions present

	A	B16; 	// Bool1 = Bool2
	JCN L83;

	L   1000;
	T   stepnumber;

L83: NOP 0;


D82: NOP 0;

//---------------------------------
// End of network: jump here if step not active
// Jump to end of this FB if the step has been active to avoid
// execution of another step in the same scan
//---------------------------------
	JU	ENDS;
J82: NOP 0;

//__phase_example_Step_990_END

NETWORK
TITLE = Step 1000
//___phase_example_Step_1000_
//================================
// function call
//================================

// skip this network if stepnumber not equal to 1000
	L 	stepnumber;
	L 	1000;
	==I;
	JCN J83;

//---------------------------------
// Actions (continuouss)
//---------------------------------

// Action: function call: write_to_DB_DW (50, 20, 123)
	CALL write_to_DB_DW
	(DB_NO := 50,
	Location := 20,
	Value := 123);

// Action: function call: write_to_DB_DW (DB_NO, 20, 123)
	CALL write_to_DB_DW
	(DB_NO := DB_NO,
	Location := 20,
	Value := 123);

// Action: function call: intvar = somefunction(34,32)
	CALL somefunction
	(arg1 := 34,
	arg2 := 32);

//---------------------------------
// --- TRANSITION TO S0 ---
//---------------------------------

// Transition Logic
	SET;	// make sure RLO is high so the transition can happen when no conditions present

	JCN L84;

	L   0;
	T   stepnumber;

L84: NOP 0;


D83: NOP 0;

//---------------------------------
// End of network: jump here if step not active
// Jump to end of this FB if the step has been active to avoid
// execution of another step in the same scan
//---------------------------------
	JU	ENDS;
J83: NOP 0;

//__phase_example_Step_1000_END





NETWORK
TITLE = Step 8000
//___phase_example_Step_8000_
//================================
// Holding
//================================

// skip this network if stepnumber not equal to 8000
	L 	stepnumber;
	L 	8000;
	==I;
	JCN J84;

//---------------------------------
// Actions (continuouss)
//---------------------------------

//---------------------------------
// --- TRANSITION TO S8990 ---
//---------------------------------

// Transition Logic
	SET;	// make sure RLO is high so the transition can happen when no conditions present

	JCN L85;

	L   8990;
	T   stepnumber;

L85: NOP 0;


D84: NOP 0;

//---------------------------------
// End of network: jump here if step not active
// Jump to end of this FB if the step has been active to avoid
// execution of another step in the same scan
//---------------------------------
	JU	ENDS;
J84: NOP 0;

//__phase_example_Step_8000_END






NETWORK
TITLE = END OF THE STEPS AND TRANSITIONS
//################################
//################################
// Placeholder network to indicate the end of the actual sequence
//################################
//################################

// jump location for the step that is currently active
ENDS:	NOP 0;


NETWORK
TITLE = Write EMs
//--------------------------------
//
//--------------------------------

	CALL FC21 (
	   EM_ID                    := EM_I_OUT_ID,
	   UDT_LOCATION             := #EM_I_OUT,
	   UDT_OFFSET               := 40,
	   Length                   := 40,
	   Request					:=EM_I_OUT.Request,
	   Owner					:=EM_I_OUT.Owner,
	   EM_addressing_error      := M      0.0,
	   RETVAL                   := MW     0);

	CALL FC21 (
	   EM_ID                    := Some_Dyn_EM_ID,
	   UDT_LOCATION             := #Some_Dyn_EM,
	   UDT_OFFSET               := 40,
	   Length                   := 40,
	   Request					:=Some_Dyn_EM.Request,
	   Owner					:=Some_Dyn_EM.Owner,
	   EM_addressing_error      := M      0.0,
	   RETVAL                   := MW     0);


END_FUNCTION_BLOCK



// <SPLIT>UNIT_INSTANCE_T100.awl</SPLIT>


// ___T100

// EM DB
//
// DB701 = T100
DATA_BLOCK "T100"

STRUCT

	Product_ID { S7_m_c := 'true' }: DINT ;	// ID of the product currently in the unit

END_STRUCT

BEGIN
END_DATA_BLOCK

FUNCTION "T100_FC" : VOID
TITLE =T100_FC
// T100_FC

AUTHOR :
FAMILY : 'unit'
NAME : namehead
VERSION : 0.1

BEGIN

NETWORK
TITLE = Main
//--------------------------------
//
//--------------------------------





END_FUNCTION


// <SPLIT>UNIT_INSTANCE_T101.awl</SPLIT>


// ___T101

// EM DB
//
// DB702 = T101
DATA_BLOCK "T101"

STRUCT

	Product_ID { S7_m_c := 'true' }: DINT ;	// ID of the product currently in the unit

END_STRUCT

BEGIN
END_DATA_BLOCK

FUNCTION "T101_FC" : VOID
TITLE =T101_FC
// T101_FC

AUTHOR :
FAMILY : 'unit'
NAME : namehead
VERSION : 0.1

BEGIN

NETWORK
TITLE = Main
//--------------------------------
//
//--------------------------------





END_FUNCTION


// <SPLIT>UNIT_INSTANCE_T102.awl</SPLIT>


// ___T102

// EM DB
//
// DB703 = T102
DATA_BLOCK "T102"

STRUCT

	Product_ID { S7_m_c := 'true' }: DINT ;	// ID of the product currently in the unit

END_STRUCT

BEGIN
END_DATA_BLOCK

FUNCTION "T102_FC" : VOID
TITLE =T102_FC
// T102_FC

AUTHOR :
FAMILY : 'unit'
NAME : namehead
VERSION : 0.1

BEGIN

NETWORK
TITLE = Main
//--------------------------------
//
//--------------------------------





END_FUNCTION


// <SPLIT>UNIT_INSTANCE_T103.awl</SPLIT>


// ___T103

// EM DB
//
// DB704 = T103
DATA_BLOCK "T103"

STRUCT

	Product_ID { S7_m_c := 'true' }: DINT ;	// ID of the product currently in the unit

END_STRUCT

BEGIN
END_DATA_BLOCK

FUNCTION "T103_FC" : VOID
TITLE =T103_FC
// T103_FC

AUTHOR :
FAMILY : 'unit'
NAME : namehead
VERSION : 0.1

BEGIN

NETWORK
TITLE = Main
//--------------------------------
//
//--------------------------------





END_FUNCTION


// <SPLIT>UNIT_INSTANCE_T104.awl</SPLIT>


// ___T104

// EM DB
//
// DB705 = T104
DATA_BLOCK "T104"

STRUCT

	Product_ID { S7_m_c := 'true' }: DINT ;	// ID of the product currently in the unit

END_STRUCT

BEGIN
END_DATA_BLOCK

FUNCTION "T104_FC" : VOID
TITLE =T104_FC
// T104_FC

AUTHOR :
FAMILY : 'unit'
NAME : namehead
VERSION : 0.1

BEGIN

NETWORK
TITLE = Main
//--------------------------------
//
//--------------------------------





END_FUNCTION


// <SPLIT>UNIT_INSTANCE_T105.awl</SPLIT>


// ___T105

// EM DB
//
// DB706 = T105
DATA_BLOCK "T105"

STRUCT

	Product_ID { S7_m_c := 'true' }: DINT ;	// ID of the product currently in the unit

END_STRUCT

BEGIN
END_DATA_BLOCK

FUNCTION "T105_FC" : VOID
TITLE =T105_FC
// T105_FC

AUTHOR :
FAMILY : 'unit'
NAME : namehead
VERSION : 0.1

BEGIN

NETWORK
TITLE = Main
//--------------------------------
//
//--------------------------------





END_FUNCTION


// <SPLIT>UNIT_INSTANCE_T106.awl</SPLIT>


// ___T106

// EM DB
//
// DB707 = T106
DATA_BLOCK "T106"

STRUCT

	Product_ID { S7_m_c := 'true' }: DINT ;	// ID of the product currently in the unit

END_STRUCT

BEGIN
END_DATA_BLOCK

FUNCTION "T106_FC" : VOID
TITLE =T106_FC
// T106_FC

AUTHOR :
FAMILY : 'unit'
NAME : namehead
VERSION : 0.1

BEGIN

NETWORK
TITLE = Main
//--------------------------------
//
//--------------------------------





END_FUNCTION


// <SPLIT>UNIT_INSTANCE_T107.awl</SPLIT>


// ___T107

// EM DB
//
// DB708 = T107
DATA_BLOCK "T107"

STRUCT

	Product_ID { S7_m_c := 'true' }: DINT ;	// ID of the product currently in the unit

END_STRUCT

BEGIN
END_DATA_BLOCK

FUNCTION "T107_FC" : VOID
TITLE =T107_FC
// T107_FC

AUTHOR :
FAMILY : 'unit'
NAME : namehead
VERSION : 0.1

BEGIN

NETWORK
TITLE = Main
//--------------------------------
//
//--------------------------------





END_FUNCTION


// <SPLIT>UNIT_INSTANCE_T108.awl</SPLIT>


// ___T108

// EM DB
//
// DB709 = T108
DATA_BLOCK "T108"

STRUCT

	Product_ID { S7_m_c := 'true' }: DINT ;	// ID of the product currently in the unit

END_STRUCT

BEGIN
END_DATA_BLOCK

FUNCTION "T108_FC" : VOID
TITLE =T108_FC
// T108_FC

AUTHOR :
FAMILY : 'unit'
NAME : namehead
VERSION : 0.1

BEGIN

NETWORK
TITLE = Main
//--------------------------------
//
//--------------------------------





END_FUNCTION


// <SPLIT>UNIT_INSTANCE_T109.awl</SPLIT>


// ___T109

// EM DB
//
// DB710 = T109
DATA_BLOCK "T109"

STRUCT

	Product_ID { S7_m_c := 'true' }: DINT ;	// ID of the product currently in the unit

END_STRUCT

BEGIN
END_DATA_BLOCK

FUNCTION "T109_FC" : VOID
TITLE =T109_FC
// T109_FC

AUTHOR :
FAMILY : 'unit'
NAME : namehead
VERSION : 0.1

BEGIN

NETWORK
TITLE = Main
//--------------------------------
//
//--------------------------------





END_FUNCTION


// <SPLIT>UNIT_INSTANCE_T110.awl</SPLIT>


// ___T110

// EM DB
//
// DB711 = T110
DATA_BLOCK "T110"

STRUCT

	Product_ID { S7_m_c := 'true' }: DINT ;	// ID of the product currently in the unit

END_STRUCT

BEGIN
END_DATA_BLOCK

FUNCTION "T110_FC" : VOID
TITLE =T110_FC
// T110_FC

AUTHOR :
FAMILY : 'unit'
NAME : namehead
VERSION : 0.1

BEGIN

NETWORK
TITLE = Main
//--------------------------------
//
//--------------------------------





END_FUNCTION


// <SPLIT>UNIT_INSTANCE_T111.awl</SPLIT>


// ___T111

// EM DB
//
// DB712 = T111
DATA_BLOCK "T111"

STRUCT

	Product_ID { S7_m_c := 'true' }: DINT ;	// ID of the product currently in the unit

END_STRUCT

BEGIN
END_DATA_BLOCK

FUNCTION "T111_FC" : VOID
TITLE =T111_FC
// T111_FC

AUTHOR :
FAMILY : 'unit'
NAME : namehead
VERSION : 0.1

BEGIN

NETWORK
TITLE = Main
//--------------------------------
//
//--------------------------------





END_FUNCTION


// <SPLIT>UNIT_INSTANCE_T112.awl</SPLIT>


// ___T112

// EM DB
//
// DB713 = T112
DATA_BLOCK "T112"

STRUCT

	Product_ID { S7_m_c := 'true' }: DINT ;	// ID of the product currently in the unit

END_STRUCT

BEGIN
END_DATA_BLOCK

FUNCTION "T112_FC" : VOID
TITLE =T112_FC
// T112_FC

AUTHOR :
FAMILY : 'unit'
NAME : namehead
VERSION : 0.1

BEGIN

NETWORK
TITLE = Main
//--------------------------------
//
//--------------------------------





END_FUNCTION


// <SPLIT>UNIT_INSTANCE_T113.awl</SPLIT>


// ___T113

// EM DB
//
// DB714 = T113
DATA_BLOCK "T113"

STRUCT

	Product_ID { S7_m_c := 'true' }: DINT ;	// ID of the product currently in the unit

END_STRUCT

BEGIN
END_DATA_BLOCK

FUNCTION "T113_FC" : VOID
TITLE =T113_FC
// T113_FC

AUTHOR :
FAMILY : 'unit'
NAME : namehead
VERSION : 0.1

BEGIN

NETWORK
TITLE = Main
//--------------------------------
//
//--------------------------------





END_FUNCTION


// <SPLIT>UNIT_INSTANCE_T114.awl</SPLIT>


// ___T114

// EM DB
//
// DB715 = T114
DATA_BLOCK "T114"

STRUCT

	Product_ID { S7_m_c := 'true' }: DINT ;	// ID of the product currently in the unit

END_STRUCT

BEGIN
END_DATA_BLOCK

FUNCTION "T114_FC" : VOID
TITLE =T114_FC
// T114_FC

AUTHOR :
FAMILY : 'unit'
NAME : namehead
VERSION : 0.1

BEGIN

NETWORK
TITLE = Main
//--------------------------------
//
//--------------------------------





END_FUNCTION


// <SPLIT>UNIT_INSTANCE_R100.awl</SPLIT>


// ___R100

// EM DB
//
// DB813 = R100
DATA_BLOCK "R100"

STRUCT

	Product_ID { S7_m_c := 'true' }: DINT ;	// ID of the product currently in the unit

END_STRUCT

BEGIN
END_DATA_BLOCK

FUNCTION "R100_FC" : VOID
TITLE =R100_FC
// R100_FC

AUTHOR :
FAMILY : 'unit'
NAME : namehead
VERSION : 0.1

BEGIN

NETWORK
TITLE = Main
//--------------------------------
//
//--------------------------------





END_FUNCTION


// <SPLIT>UNIT_INSTANCE_R101.awl</SPLIT>


// ___R101

// EM DB
//
// DB814 = R101
DATA_BLOCK "R101"

STRUCT

	Product_ID { S7_m_c := 'true' }: DINT ;	// ID of the product currently in the unit

END_STRUCT

BEGIN
END_DATA_BLOCK

FUNCTION "R101_FC" : VOID
TITLE =R101_FC
// R101_FC

AUTHOR :
FAMILY : 'unit'
NAME : namehead
VERSION : 0.1

BEGIN

NETWORK
TITLE = Main
//--------------------------------
//
//--------------------------------





END_FUNCTION



// <SPLIT>CM_INSTANCE_XV001.awl</SPLIT>


// ___XV001

// CM Instance DB
// DB732 = XV001
// FB630 = BST_VALVE_400
DATA_BLOCK DB732 FB630
BEGIN
END_DATA_BLOCK

FUNCTION "XV001_FC" : VOID
TITLE =XV001_FC
// XV001_FC
// Some Valve  on drawing 1
AUTHOR :
FAMILY : 'cminst'
NAME : namehead
VERSION : 0.1

BEGIN

NETWORK
TITLE = Main
//--------------------------------
// PLC1
//--------------------------------

CALL FB630, DB 732;

END_FUNCTION


// <SPLIT>CM_INSTANCE_XV002.awl</SPLIT>


// ___XV002

// CM Instance DB
// DB733 = XV002
// FB630 = BST_VALVE_400
DATA_BLOCK DB733 FB630
BEGIN
END_DATA_BLOCK

FUNCTION "XV002_FC" : VOID
TITLE =XV002_FC
// XV002_FC
// Some Valve  on drawing 2
AUTHOR :
FAMILY : 'cminst'
NAME : namehead
VERSION : 0.1

BEGIN

NETWORK
TITLE = Main
//--------------------------------
// PLC1
//--------------------------------

CALL FB630, DB 733;

END_FUNCTION


// <SPLIT>CM_INSTANCE_XV003.awl</SPLIT>


// ___XV003

// CM Instance DB
// DB734 = XV003
// FB630 = BST_VALVE_400
DATA_BLOCK DB734 FB630
BEGIN
END_DATA_BLOCK

FUNCTION "XV003_FC" : VOID
TITLE =XV003_FC
// XV003_FC
// Some Valve  on drawing 3
AUTHOR :
FAMILY : 'cminst'
NAME : namehead
VERSION : 0.1

BEGIN

NETWORK
TITLE = Main
//--------------------------------
// PLC1
//--------------------------------

CALL FB630, DB 734;

END_FUNCTION


// <SPLIT>CM_INSTANCE_XV004.awl</SPLIT>


// ___XV004

// CM Instance DB
// DB735 = XV004
// FB630 = BST_VALVE_400
DATA_BLOCK DB735 FB630
BEGIN
END_DATA_BLOCK

FUNCTION "XV004_FC" : VOID
TITLE =XV004_FC
// XV004_FC
// Some Valve  on drawing 4
AUTHOR :
FAMILY : 'cminst'
NAME : namehead
VERSION : 0.1

BEGIN

NETWORK
TITLE = Main
//--------------------------------
// PLC1
//--------------------------------

CALL FB630, DB 735;

END_FUNCTION












// <SPLIT>CM_INSTANCE_XV300.awl</SPLIT>


// ___XV300

// CM Instance DB
// DB746 = XV300
// FB630 = BST_VALVE_400
DATA_BLOCK DB746 FB630
BEGIN
END_DATA_BLOCK

FUNCTION "XV300_FC" : VOID
TITLE =XV300_FC
// XV300_FC
// Some Valve  on drawing 15
AUTHOR :
FAMILY : 'cminst'
NAME : namehead
VERSION : 0.1

BEGIN

NETWORK
TITLE = Main
//--------------------------------
// PLC1
//--------------------------------

CALL FB630, DB 746;

END_FUNCTION


// <SPLIT>CM_INSTANCE_XV400.awl</SPLIT>


// ___XV400

// CM Instance DB
// DB747 = XV400
// FB630 = BST_VALVE_400
DATA_BLOCK DB747 FB630
BEGIN
END_DATA_BLOCK

FUNCTION "XV400_FC" : VOID
TITLE =XV400_FC
// XV400_FC
// Some Valve  on drawing 16
AUTHOR :
FAMILY : 'cminst'
NAME : namehead
VERSION : 0.1

BEGIN

NETWORK
TITLE = Main
//--------------------------------
// PLC1
//--------------------------------

CALL FB630, DB 747;

END_FUNCTION


// <SPLIT>CM_INSTANCE_XV500.awl</SPLIT>


// ___XV500

// CM Instance DB
// DB748 = XV500
// FB630 = BST_VALVE_400
DATA_BLOCK DB748 FB630
BEGIN
END_DATA_BLOCK

FUNCTION "XV500_FC" : VOID
TITLE =XV500_FC
// XV500_FC
// Some Valve  on drawing 17
AUTHOR :
FAMILY : 'cminst'
NAME : namehead
VERSION : 0.1

BEGIN

NETWORK
TITLE = Main
//--------------------------------
// PLC1
//--------------------------------

CALL FB630, DB 748;

END_FUNCTION


// <SPLIT>CM_INSTANCE_XV301.awl</SPLIT>


// ___XV301

// CM Instance DB
// DB749 = XV301
// FB630 = BST_VALVE_400
DATA_BLOCK DB749 FB630
BEGIN
END_DATA_BLOCK

FUNCTION "XV301_FC" : VOID
TITLE =XV301_FC
// XV301_FC
// Some Valve  on drawing 18
AUTHOR :
FAMILY : 'cminst'
NAME : namehead
VERSION : 0.1

BEGIN

NETWORK
TITLE = Main
//--------------------------------
// PLC1
//--------------------------------

CALL FB630, DB 749;

END_FUNCTION



// <SPLIT>CM_INSTANCE_XV501.awl</SPLIT>


// ___XV501

// CM Instance DB
// DB751 = XV501
// FB630 = BST_VALVE_400
DATA_BLOCK DB751 FB630
BEGIN
END_DATA_BLOCK

FUNCTION "XV501_FC" : VOID
TITLE =XV501_FC
// XV501_FC
// Some Valve  on drawing 20
AUTHOR :
FAMILY : 'cminst'
NAME : namehead
VERSION : 0.1

BEGIN

NETWORK
TITLE = Main
//--------------------------------
// PLC1
//--------------------------------

CALL FB630, DB 751;

END_FUNCTION


// <SPLIT>CM_INSTANCE_XV401.awl</SPLIT>


// ___XV401

// CM Instance DB
// DB752 = XV401
// FB630 = BST_VALVE_400
DATA_BLOCK DB752 FB630
BEGIN
END_DATA_BLOCK

FUNCTION "XV401_FC" : VOID
TITLE =XV401_FC
// XV401_FC
// Some Valve  on drawing 21
AUTHOR :
FAMILY : 'cminst'
NAME : namehead
VERSION : 0.1

BEGIN

NETWORK
TITLE = Main
//--------------------------------
// PLC1
//--------------------------------

CALL FB630, DB 752;

END_FUNCTION


// <SPLIT>CM_INSTANCE_MV001.awl</SPLIT>


// ___MV001

// CM Instance DB
// DB753 = MV001
// FB630 = BST_VALVE_400
DATA_BLOCK DB753 FB630
BEGIN
END_DATA_BLOCK

FUNCTION "MV001_FC" : VOID
TITLE =MV001_FC
// MV001_FC

AUTHOR :
FAMILY : 'cminst'
NAME : namehead
VERSION : 0.1

BEGIN

NETWORK
TITLE = Main
//--------------------------------
// PLC1
//--------------------------------

CALL FB630, DB 753;

END_FUNCTION


// <SPLIT>CM_INSTANCE_MV002.awl</SPLIT>


// ___MV002

// CM Instance DB
// DB754 = MV002
// FB630 = BST_VALVE_400
DATA_BLOCK DB754 FB630
BEGIN
END_DATA_BLOCK

FUNCTION "MV002_FC" : VOID
TITLE =MV002_FC
// MV002_FC

AUTHOR :
FAMILY : 'cminst'
NAME : namehead
VERSION : 0.1

BEGIN

NETWORK
TITLE = Main
//--------------------------------
// PLC1
//--------------------------------

CALL FB630, DB 754;

END_FUNCTION


// <SPLIT>CM_INSTANCE_MV003.awl</SPLIT>


// ___MV003

// CM Instance DB
// DB755 = MV003
// FB630 = BST_VALVE_400
DATA_BLOCK DB755 FB630
BEGIN
END_DATA_BLOCK

FUNCTION "MV003_FC" : VOID
TITLE =MV003_FC
// MV003_FC

AUTHOR :
FAMILY : 'cminst'
NAME : namehead
VERSION : 0.1

BEGIN

NETWORK
TITLE = Main
//--------------------------------
// PLC1
//--------------------------------

CALL FB630, DB 755;

END_FUNCTION


// <SPLIT>CM_INSTANCE_MV004.awl</SPLIT>


// ___MV004

// CM Instance DB
// DB756 = MV004
// FB630 = BST_VALVE_400
DATA_BLOCK DB756 FB630
BEGIN
END_DATA_BLOCK

FUNCTION "MV004_FC" : VOID
TITLE =MV004_FC
// MV004_FC

AUTHOR :
FAMILY : 'cminst'
NAME : namehead
VERSION : 0.1

BEGIN

NETWORK
TITLE = Main
//--------------------------------
// PLC1
//--------------------------------

CALL FB630, DB 756;

END_FUNCTION


// <SPLIT>CM_INSTANCE_MV005.awl</SPLIT>


// ___MV005

// CM Instance DB
// DB757 = MV005
// FB630 = BST_VALVE_400
DATA_BLOCK DB757 FB630
BEGIN
END_DATA_BLOCK

FUNCTION "MV005_FC" : VOID
TITLE =MV005_FC
// MV005_FC

AUTHOR :
FAMILY : 'cminst'
NAME : namehead
VERSION : 0.1

BEGIN

NETWORK
TITLE = Main
//--------------------------------
// PLC1
//--------------------------------

CALL FB630, DB 757;

END_FUNCTION


// <SPLIT>CM_INSTANCE_MV006.awl</SPLIT>


// ___MV006

// CM Instance DB
// DB758 = MV006
// FB630 = BST_VALVE_400
DATA_BLOCK DB758 FB630
BEGIN
END_DATA_BLOCK

FUNCTION "MV006_FC" : VOID
TITLE =MV006_FC
// MV006_FC

AUTHOR :
FAMILY : 'cminst'
NAME : namehead
VERSION : 0.1

BEGIN

NETWORK
TITLE = Main
//--------------------------------
// PLC1
//--------------------------------

CALL FB630, DB 758;

END_FUNCTION


// <SPLIT>CM_INSTANCE_MV007.awl</SPLIT>


// ___MV007

// CM Instance DB
// DB759 = MV007
// FB630 = BST_VALVE_400
DATA_BLOCK DB759 FB630
BEGIN
END_DATA_BLOCK

FUNCTION "MV007_FC" : VOID
TITLE =MV007_FC
// MV007_FC

AUTHOR :
FAMILY : 'cminst'
NAME : namehead
VERSION : 0.1

BEGIN

NETWORK
TITLE = Main
//--------------------------------
// PLC1
//--------------------------------

CALL FB630, DB 759;

END_FUNCTION









// <SPLIT>CM_INSTANCE_P100.awl</SPLIT>


// ___P100

// CM Instance DB
// DB767 = P100
// FB680 = BST_MOTOR_400
DATA_BLOCK DB767 FB680
BEGIN
END_DATA_BLOCK

FUNCTION "P100_FC" : VOID
TITLE =P100_FC
// P100_FC

AUTHOR :
FAMILY : 'cminst'
NAME : namehead
VERSION : 0.1

BEGIN

NETWORK
TITLE = Main
//--------------------------------
// PLC1
//--------------------------------

CALL FB680, DB 767;

END_FUNCTION


// <SPLIT>CM_INSTANCE_P200.awl</SPLIT>


// ___P200

// CM Instance DB
// DB768 = P200
// FB680 = BST_MOTOR_400
DATA_BLOCK DB768 FB680
BEGIN
END_DATA_BLOCK

FUNCTION "P200_FC" : VOID
TITLE =P200_FC
// P200_FC

AUTHOR :
FAMILY : 'cminst'
NAME : namehead
VERSION : 0.1

BEGIN

NETWORK
TITLE = Main
//--------------------------------
// PLC1
//--------------------------------

CALL FB680, DB 768;

END_FUNCTION


// <SPLIT>CM_INSTANCE_P101.awl</SPLIT>


// ___P101

// CM Instance DB
// DB769 = P101
// FB680 = BST_MOTOR_400
DATA_BLOCK DB769 FB680
BEGIN
END_DATA_BLOCK

FUNCTION "P101_FC" : VOID
TITLE =P101_FC
// P101_FC

AUTHOR :
FAMILY : 'cminst'
NAME : namehead
VERSION : 0.1

BEGIN

NETWORK
TITLE = Main
//--------------------------------
// PLC1
//--------------------------------

CALL FB680, DB 769;

END_FUNCTION


// <SPLIT>CM_INSTANCE_P201.awl</SPLIT>


// ___P201

// CM Instance DB
// DB770 = P201
// FB680 = BST_MOTOR_400
DATA_BLOCK DB770 FB680
BEGIN
END_DATA_BLOCK

FUNCTION "P201_FC" : VOID
TITLE =P201_FC
// P201_FC

AUTHOR :
FAMILY : 'cminst'
NAME : namehead
VERSION : 0.1

BEGIN

NETWORK
TITLE = Main
//--------------------------------
// PLC1
//--------------------------------

CALL FB680, DB 770;

END_FUNCTION


// <SPLIT>CM_INSTANCE_M100.awl</SPLIT>


// ___M100

// CM Instance DB
// DB771 = M100
// FB680 = BST_SINAG120_400
DATA_BLOCK DB771 FB680
BEGIN
END_DATA_BLOCK

FUNCTION "M100_FC" : VOID
TITLE =M100_FC
// M100_FC

AUTHOR :
FAMILY : 'cminst'
NAME : namehead
VERSION : 0.1

BEGIN

NETWORK
TITLE = Main
//--------------------------------
// PLC1
//--------------------------------

CALL FB680, DB 771;

END_FUNCTION


// <SPLIT>CM_INSTANCE_M101.awl</SPLIT>


// ___M101

// CM Instance DB
// DB772 = M101
// FB680 = BST_SINAG120_400
DATA_BLOCK DB772 FB680
BEGIN
END_DATA_BLOCK

FUNCTION "M101_FC" : VOID
TITLE =M101_FC
// M101_FC

AUTHOR :
FAMILY : 'cminst'
NAME : namehead
VERSION : 0.1

BEGIN

NETWORK
TITLE = Main
//--------------------------------
// PLC1
//--------------------------------

CALL FB680, DB 772;

END_FUNCTION


// <SPLIT>CM_INSTANCE_M102.awl</SPLIT>


// ___M102

// CM Instance DB
// DB773 = M102
// FB680 = BST_SINAG120_400
DATA_BLOCK DB773 FB680
BEGIN
END_DATA_BLOCK

FUNCTION "M102_FC" : VOID
TITLE =M102_FC
// M102_FC

AUTHOR :
FAMILY : 'cminst'
NAME : namehead
VERSION : 0.1

BEGIN

NETWORK
TITLE = Main
//--------------------------------
// PLC1
//--------------------------------

CALL FB680, DB 773;

END_FUNCTION


// <SPLIT>CM_INSTANCE_M103.awl</SPLIT>


// ___M103

// CM Instance DB
// DB774 = M103
// FB680 = BST_SINAG120_400
DATA_BLOCK DB774 FB680
BEGIN
END_DATA_BLOCK

FUNCTION "M103_FC" : VOID
TITLE =M103_FC
// M103_FC

AUTHOR :
FAMILY : 'cminst'
NAME : namehead
VERSION : 0.1

BEGIN

NETWORK
TITLE = Main
//--------------------------------
// PLC1
//--------------------------------

CALL FB680, DB 774;

END_FUNCTION


// <SPLIT>CM_INSTANCE_M104.awl</SPLIT>


// ___M104

// CM Instance DB
// DB775 = M104
// FB680 = BST_SINAG120_400
DATA_BLOCK DB775 FB680
BEGIN
END_DATA_BLOCK

FUNCTION "M104_FC" : VOID
TITLE =M104_FC
// M104_FC

AUTHOR :
FAMILY : 'cminst'
NAME : namehead
VERSION : 0.1

BEGIN

NETWORK
TITLE = Main
//--------------------------------
// PLC1
//--------------------------------

CALL FB680, DB 775;

END_FUNCTION


// <SPLIT>CM_INSTANCE_M105.awl</SPLIT>


// ___M105

// CM Instance DB
// DB776 = M105
// FB680 = BST_SINAG120_400
DATA_BLOCK DB776 FB680
BEGIN
END_DATA_BLOCK

FUNCTION "M105_FC" : VOID
TITLE =M105_FC
// M105_FC

AUTHOR :
FAMILY : 'cminst'
NAME : namehead
VERSION : 0.1

BEGIN

NETWORK
TITLE = Main
//--------------------------------
// PLC1
//--------------------------------

CALL FB680, DB 776;

END_FUNCTION


// <SPLIT>CM_INSTANCE_M106.awl</SPLIT>


// ___M106

// CM Instance DB
// DB777 = M106
// FB680 = BST_SINAG120_400
DATA_BLOCK DB777 FB680
BEGIN
END_DATA_BLOCK

FUNCTION "M106_FC" : VOID
TITLE =M106_FC
// M106_FC

AUTHOR :
FAMILY : 'cminst'
NAME : namehead
VERSION : 0.1

BEGIN

NETWORK
TITLE = Main
//--------------------------------
// PLC1
//--------------------------------

CALL FB680, DB 777;

END_FUNCTION


// <SPLIT>CM_INSTANCE_LT001.awl</SPLIT>


// ___LT001

// CM Instance DB
// DB778 = LT001
// FB640 = BST_ANALOG_400
DATA_BLOCK DB778 FB640
BEGIN
END_DATA_BLOCK

FUNCTION "LT001_FC" : VOID
TITLE =LT001_FC
// LT001_FC

AUTHOR :
FAMILY : 'cminst'
NAME : namehead
VERSION : 0.1

BEGIN

NETWORK
TITLE = Main
//--------------------------------
// PLC1
//--------------------------------

CALL FB640, DB 778;

END_FUNCTION


// <SPLIT>CM_INSTANCE_LT002.awl</SPLIT>


// ___LT002

// CM Instance DB
// DB779 = LT002
// FB640 = BST_ANALOG_400
DATA_BLOCK DB779 FB640
BEGIN
END_DATA_BLOCK

FUNCTION "LT002_FC" : VOID
TITLE =LT002_FC
// LT002_FC

AUTHOR :
FAMILY : 'cminst'
NAME : namehead
VERSION : 0.1

BEGIN

NETWORK
TITLE = Main
//--------------------------------
// PLC1
//--------------------------------

CALL FB640, DB 779;

END_FUNCTION


// <SPLIT>CM_INSTANCE_LT003.awl</SPLIT>


// ___LT003

// CM Instance DB
// DB780 = LT003
// FB640 = BST_ANALOG_400
DATA_BLOCK DB780 FB640
BEGIN
END_DATA_BLOCK

FUNCTION "LT003_FC" : VOID
TITLE =LT003_FC
// LT003_FC

AUTHOR :
FAMILY : 'cminst'
NAME : namehead
VERSION : 0.1

BEGIN

NETWORK
TITLE = Main
//--------------------------------
// PLC1
//--------------------------------

CALL FB640, DB 780;

END_FUNCTION


// <SPLIT>CM_INSTANCE_LT004.awl</SPLIT>


// ___LT004

// CM Instance DB
// DB781 = LT004
// FB640 = BST_ANALOG_400
DATA_BLOCK DB781 FB640
BEGIN
END_DATA_BLOCK

FUNCTION "LT004_FC" : VOID
TITLE =LT004_FC
// LT004_FC

AUTHOR :
FAMILY : 'cminst'
NAME : namehead
VERSION : 0.1

BEGIN

NETWORK
TITLE = Main
//--------------------------------
// PLC1
//--------------------------------

CALL FB640, DB 781;

END_FUNCTION


// <SPLIT>CM_INSTANCE_LT005.awl</SPLIT>


// ___LT005

// CM Instance DB
// DB782 = LT005
// FB640 = BST_ANALOG_400
DATA_BLOCK DB782 FB640
BEGIN
END_DATA_BLOCK

FUNCTION "LT005_FC" : VOID
TITLE =LT005_FC
// LT005_FC

AUTHOR :
FAMILY : 'cminst'
NAME : namehead
VERSION : 0.1

BEGIN

NETWORK
TITLE = Main
//--------------------------------
// PLC1
//--------------------------------

CALL FB640, DB 782;

END_FUNCTION


// <SPLIT>CM_INSTANCE_LT006.awl</SPLIT>


// ___LT006

// CM Instance DB
// DB783 = LT006
// FB640 = BST_ANALOG_400
DATA_BLOCK DB783 FB640
BEGIN
END_DATA_BLOCK

FUNCTION "LT006_FC" : VOID
TITLE =LT006_FC
// LT006_FC

AUTHOR :
FAMILY : 'cminst'
NAME : namehead
VERSION : 0.1

BEGIN

NETWORK
TITLE = Main
//--------------------------------
// PLC1
//--------------------------------

CALL FB640, DB 783;

END_FUNCTION


// <SPLIT>CM_INSTANCE_LT007.awl</SPLIT>


// ___LT007

// CM Instance DB
// DB784 = LT007
// FB640 = BST_ANALOG_400
DATA_BLOCK DB784 FB640
BEGIN
END_DATA_BLOCK

FUNCTION "LT007_FC" : VOID
TITLE =LT007_FC
// LT007_FC

AUTHOR :
FAMILY : 'cminst'
NAME : namehead
VERSION : 0.1

BEGIN

NETWORK
TITLE = Main
//--------------------------------
// PLC1
//--------------------------------

CALL FB640, DB 784;

END_FUNCTION


// <SPLIT>CM_INSTANCE_LT100.awl</SPLIT>


// ___LT100

// CM Instance DB
// DB785 = LT100
// FB640 = BST_ANALOG_400
DATA_BLOCK DB785 FB640
BEGIN
END_DATA_BLOCK

FUNCTION "LT100_FC" : VOID
TITLE =LT100_FC
// LT100_FC

AUTHOR :
FAMILY : 'cminst'
NAME : namehead
VERSION : 0.1

BEGIN

NETWORK
TITLE = Main
//--------------------------------
// PLC1
//--------------------------------

CALL FB640, DB 785;

END_FUNCTION


// <SPLIT>CM_INSTANCE_LT200.awl</SPLIT>


// ___LT200

// CM Instance DB
// DB786 = LT200
// FB640 = BST_ANALOG_400
DATA_BLOCK DB786 FB640
BEGIN
END_DATA_BLOCK

FUNCTION "LT200_FC" : VOID
TITLE =LT200_FC
// LT200_FC

AUTHOR :
FAMILY : 'cminst'
NAME : namehead
VERSION : 0.1

BEGIN

NETWORK
TITLE = Main
//--------------------------------
// PLC1
//--------------------------------

CALL FB640, DB 786;

END_FUNCTION


// <SPLIT>CM_INSTANCE_LT101.awl</SPLIT>


// ___LT101

// CM Instance DB
// DB787 = LT101
// FB640 = BST_ANALOG_400
DATA_BLOCK DB787 FB640
BEGIN
END_DATA_BLOCK

FUNCTION "LT101_FC" : VOID
TITLE =LT101_FC
// LT101_FC

AUTHOR :
FAMILY : 'cminst'
NAME : namehead
VERSION : 0.1

BEGIN

NETWORK
TITLE = Main
//--------------------------------
// PLC1
//--------------------------------

CALL FB640, DB 787;

END_FUNCTION


// <SPLIT>CM_INSTANCE_LT201.awl</SPLIT>


// ___LT201

// CM Instance DB
// DB788 = LT201
// FB640 = BST_ANALOG_400
DATA_BLOCK DB788 FB640
BEGIN
END_DATA_BLOCK

FUNCTION "LT201_FC" : VOID
TITLE =LT201_FC
// LT201_FC

AUTHOR :
FAMILY : 'cminst'
NAME : namehead
VERSION : 0.1

BEGIN

NETWORK
TITLE = Main
//--------------------------------
// PLC1
//--------------------------------

CALL FB640, DB 788;

END_FUNCTION


// <SPLIT>CM_INSTANCE_LS001.awl</SPLIT>


// ___LS001

// CM Instance DB
// DB789 = LS001
// FB650 = BST_DIGITAL_400
DATA_BLOCK DB789 FB650
BEGIN
END_DATA_BLOCK

FUNCTION "LS001_FC" : VOID
TITLE =LS001_FC
// LS001_FC

AUTHOR :
FAMILY : 'cminst'
NAME : namehead
VERSION : 0.1

BEGIN

NETWORK
TITLE = Main
//--------------------------------
// PLC1
//--------------------------------

CALL FB650, DB 789;

END_FUNCTION


// <SPLIT>CM_INSTANCE_LS002.awl</SPLIT>


// ___LS002

// CM Instance DB
// DB790 = LS002
// FB650 = BST_DIGITAL_400
DATA_BLOCK DB790 FB650
BEGIN
END_DATA_BLOCK

FUNCTION "LS002_FC" : VOID
TITLE =LS002_FC
// LS002_FC

AUTHOR :
FAMILY : 'cminst'
NAME : namehead
VERSION : 0.1

BEGIN

NETWORK
TITLE = Main
//--------------------------------
// PLC1
//--------------------------------

CALL FB650, DB 790;

END_FUNCTION






// <SPLIT>CM_INSTANCE_LIC001.awl</SPLIT>


// ___LIC001

// CM Instance DB
// DB795 = LIC001
// FB670 = BST_PIDAIN_400
DATA_BLOCK DB795 FB670
BEGIN
END_DATA_BLOCK

DATA_BLOCK  DB796
// tagstruct_name = PID_interface
STRUCT
	Operator_Setpoint { S7_m_c := 'true' } : REAL;
	Set_SP { S7_m_c := 'true' } : BOOL;
	Output_Value { S7_m_c := 'true' } : REAL;
	Set_Output { S7_m_c := 'true' } : BOOL;
END_STRUCT
BEGIN
END_DATA_BLOCK

FUNCTION "LIC001_FC" : VOID
TITLE =LIC001_FC
// LIC001_FC

AUTHOR :
FAMILY : 'cminst'
NAME : namehead
VERSION : 0.1

BEGIN
NETWORK
TITLE = Change PID Setpoints
//--------------------------------
// The phase FBs write on the operator setpoints of the PID-controller
// To avoid that the setpoints are always overwritten (and blocking operator control)
// we use pulses generated by the phase to set the setpoints only at specific moments
// i_fOCmdSP (setpoint)
// i_fOCmdMANOP (output)
//--------------------------------

// Write the Operator_Setpoint
A	DB796.Set_SP;
JCN J001;

	L DB796.Operator_Setpoint;
	T DB795.i_fOCmdSP;

J001: NOP 0;


// Write the Output_Value
A	DB796.Set_Output;
JCN J002;

	L DB796.Output_Value;
	T DB795.i_fOCmdMANOP;

J002: NOP 0;

NETWORK
TITLE = Main
//--------------------------------
// PLC1
//--------------------------------

CALL FB670, DB 795;

END_FUNCTION


// <SPLIT>CM_INSTANCE_LIC002.awl</SPLIT>


// ___LIC002

// CM Instance DB
// DB797 = LIC002
// FB670 = BST_PIDAIN_400
DATA_BLOCK DB797 FB670
BEGIN
END_DATA_BLOCK

DATA_BLOCK  DB798
// tagstruct_name = PID_interface
STRUCT
	Operator_Setpoint { S7_m_c := 'true' } : REAL;
	Set_SP { S7_m_c := 'true' } : BOOL;
	Output_Value { S7_m_c := 'true' } : REAL;
	Set_Output { S7_m_c := 'true' } : BOOL;
END_STRUCT
BEGIN
END_DATA_BLOCK

FUNCTION "LIC002_FC" : VOID
TITLE =LIC002_FC
// LIC002_FC

AUTHOR :
FAMILY : 'cminst'
NAME : namehead
VERSION : 0.1

BEGIN
NETWORK
TITLE = Change PID Setpoints
//--------------------------------
// The phase FBs write on the operator setpoints of the PID-controller
// To avoid that the setpoints are always overwritten (and blocking operator control)
// we use pulses generated by the phase to set the setpoints only at specific moments
// i_fOCmdSP (setpoint)
// i_fOCmdMANOP (output)
//--------------------------------

// Write the Operator_Setpoint
A	DB798.Set_SP;
JCN J001;

	L DB798.Operator_Setpoint;
	T DB797.i_fOCmdSP;

J001: NOP 0;


// Write the Output_Value
A	DB798.Set_Output;
JCN J002;

	L DB798.Output_Value;
	T DB797.i_fOCmdMANOP;

J002: NOP 0;

NETWORK
TITLE = Main
//--------------------------------
// PLC1
//--------------------------------

CALL FB670, DB 797;

END_FUNCTION


// <SPLIT>CM_INSTANCE_LIC003.awl</SPLIT>


// ___LIC003

// CM Instance DB
// DB799 = LIC003
// FB670 = BST_PIDAIN_400
DATA_BLOCK DB799 FB670
BEGIN
END_DATA_BLOCK

DATA_BLOCK  DB800
// tagstruct_name = PID_interface
STRUCT
	Operator_Setpoint { S7_m_c := 'true' } : REAL;
	Set_SP { S7_m_c := 'true' } : BOOL;
	Output_Value { S7_m_c := 'true' } : REAL;
	Set_Output { S7_m_c := 'true' } : BOOL;
END_STRUCT
BEGIN
END_DATA_BLOCK

FUNCTION "LIC003_FC" : VOID
TITLE =LIC003_FC
// LIC003_FC

AUTHOR :
FAMILY : 'cminst'
NAME : namehead
VERSION : 0.1

BEGIN
NETWORK
TITLE = Change PID Setpoints
//--------------------------------
// The phase FBs write on the operator setpoints of the PID-controller
// To avoid that the setpoints are always overwritten (and blocking operator control)
// we use pulses generated by the phase to set the setpoints only at specific moments
// i_fOCmdSP (setpoint)
// i_fOCmdMANOP (output)
//--------------------------------

// Write the Operator_Setpoint
A	DB800.Set_SP;
JCN J001;

	L DB800.Operator_Setpoint;
	T DB799.i_fOCmdSP;

J001: NOP 0;


// Write the Output_Value
A	DB800.Set_Output;
JCN J002;

	L DB800.Output_Value;
	T DB799.i_fOCmdMANOP;

J002: NOP 0;

NETWORK
TITLE = Main
//--------------------------------
// PLC1
//--------------------------------

CALL FB670, DB 799;

END_FUNCTION


// <SPLIT>CM_INSTANCE_LIC004.awl</SPLIT>


// ___LIC004

// CM Instance DB
// DB801 = LIC004
// FB670 = BST_PIDAIN_400
DATA_BLOCK DB801 FB670
BEGIN
END_DATA_BLOCK

DATA_BLOCK  DB802
// tagstruct_name = PID_interface
STRUCT
	Operator_Setpoint { S7_m_c := 'true' } : REAL;
	Set_SP { S7_m_c := 'true' } : BOOL;
	Output_Value { S7_m_c := 'true' } : REAL;
	Set_Output { S7_m_c := 'true' } : BOOL;
END_STRUCT
BEGIN
END_DATA_BLOCK

FUNCTION "LIC004_FC" : VOID
TITLE =LIC004_FC
// LIC004_FC

AUTHOR :
FAMILY : 'cminst'
NAME : namehead
VERSION : 0.1

BEGIN
NETWORK
TITLE = Change PID Setpoints
//--------------------------------
// The phase FBs write on the operator setpoints of the PID-controller
// To avoid that the setpoints are always overwritten (and blocking operator control)
// we use pulses generated by the phase to set the setpoints only at specific moments
// i_fOCmdSP (setpoint)
// i_fOCmdMANOP (output)
//--------------------------------

// Write the Operator_Setpoint
A	DB802.Set_SP;
JCN J001;

	L DB802.Operator_Setpoint;
	T DB801.i_fOCmdSP;

J001: NOP 0;


// Write the Output_Value
A	DB802.Set_Output;
JCN J002;

	L DB802.Output_Value;
	T DB801.i_fOCmdMANOP;

J002: NOP 0;

NETWORK
TITLE = Main
//--------------------------------
// PLC1
//--------------------------------

CALL FB670, DB 801;

END_FUNCTION


// <SPLIT>CM_INSTANCE_LIC005.awl</SPLIT>


// ___LIC005

// CM Instance DB
// DB803 = LIC005
// FB670 = BST_PIDAIN_400
DATA_BLOCK DB803 FB670
BEGIN
END_DATA_BLOCK

DATA_BLOCK  DB804
// tagstruct_name = PID_interface
STRUCT
	Operator_Setpoint { S7_m_c := 'true' } : REAL;
	Set_SP { S7_m_c := 'true' } : BOOL;
	Output_Value { S7_m_c := 'true' } : REAL;
	Set_Output { S7_m_c := 'true' } : BOOL;
END_STRUCT
BEGIN
END_DATA_BLOCK

FUNCTION "LIC005_FC" : VOID
TITLE =LIC005_FC
// LIC005_FC

AUTHOR :
FAMILY : 'cminst'
NAME : namehead
VERSION : 0.1

BEGIN
NETWORK
TITLE = Change PID Setpoints
//--------------------------------
// The phase FBs write on the operator setpoints of the PID-controller
// To avoid that the setpoints are always overwritten (and blocking operator control)
// we use pulses generated by the phase to set the setpoints only at specific moments
// i_fOCmdSP (setpoint)
// i_fOCmdMANOP (output)
//--------------------------------

// Write the Operator_Setpoint
A	DB804.Set_SP;
JCN J001;

	L DB804.Operator_Setpoint;
	T DB803.i_fOCmdSP;

J001: NOP 0;


// Write the Output_Value
A	DB804.Set_Output;
JCN J002;

	L DB804.Output_Value;
	T DB803.i_fOCmdMANOP;

J002: NOP 0;

NETWORK
TITLE = Main
//--------------------------------
// PLC1
//--------------------------------

CALL FB670, DB 803;

END_FUNCTION


// <SPLIT>CM_INSTANCE_LIC006.awl</SPLIT>


// ___LIC006

// CM Instance DB
// DB805 = LIC006
// FB670 = BST_PIDAIN_400
DATA_BLOCK DB805 FB670
BEGIN
END_DATA_BLOCK

DATA_BLOCK  DB806
// tagstruct_name = PID_interface
STRUCT
	Operator_Setpoint { S7_m_c := 'true' } : REAL;
	Set_SP { S7_m_c := 'true' } : BOOL;
	Output_Value { S7_m_c := 'true' } : REAL;
	Set_Output { S7_m_c := 'true' } : BOOL;
END_STRUCT
BEGIN
END_DATA_BLOCK

FUNCTION "LIC006_FC" : VOID
TITLE =LIC006_FC
// LIC006_FC

AUTHOR :
FAMILY : 'cminst'
NAME : namehead
VERSION : 0.1

BEGIN
NETWORK
TITLE = Change PID Setpoints
//--------------------------------
// The phase FBs write on the operator setpoints of the PID-controller
// To avoid that the setpoints are always overwritten (and blocking operator control)
// we use pulses generated by the phase to set the setpoints only at specific moments
// i_fOCmdSP (setpoint)
// i_fOCmdMANOP (output)
//--------------------------------

// Write the Operator_Setpoint
A	DB806.Set_SP;
JCN J001;

	L DB806.Operator_Setpoint;
	T DB805.i_fOCmdSP;

J001: NOP 0;


// Write the Output_Value
A	DB806.Set_Output;
JCN J002;

	L DB806.Output_Value;
	T DB805.i_fOCmdMANOP;

J002: NOP 0;

NETWORK
TITLE = Main
//--------------------------------
// PLC1
//--------------------------------

CALL FB670, DB 805;

END_FUNCTION



// <SPLIT>CM_INSTANCE_FIC100.awl</SPLIT>


// ___FIC100

// CM Instance DB
// DB809 = FIC100
// FB670 = BST_PIDAIN_400
DATA_BLOCK DB809 FB670
BEGIN
END_DATA_BLOCK

DATA_BLOCK  DB810
// tagstruct_name = PID_interface
STRUCT
	Operator_Setpoint { S7_m_c := 'true' } : REAL;
	Set_SP { S7_m_c := 'true' } : BOOL;
	Output_Value { S7_m_c := 'true' } : REAL;
	Set_Output { S7_m_c := 'true' } : BOOL;
END_STRUCT
BEGIN
END_DATA_BLOCK

FUNCTION "FIC100_FC" : VOID
TITLE =FIC100_FC
// FIC100_FC

AUTHOR :
FAMILY : 'cminst'
NAME : namehead
VERSION : 0.1

BEGIN
NETWORK
TITLE = Change PID Setpoints
//--------------------------------
// The phase FBs write on the operator setpoints of the PID-controller
// To avoid that the setpoints are always overwritten (and blocking operator control)
// we use pulses generated by the phase to set the setpoints only at specific moments
// i_fOCmdSP (setpoint)
// i_fOCmdMANOP (output)
//--------------------------------

// Write the Operator_Setpoint
A	DB810.Set_SP;
JCN J001;

	L DB810.Operator_Setpoint;
	T DB809.i_fOCmdSP;

J001: NOP 0;


// Write the Output_Value
A	DB810.Set_Output;
JCN J002;

	L DB810.Output_Value;
	T DB809.i_fOCmdMANOP;

J002: NOP 0;

NETWORK
TITLE = Main
//--------------------------------
// PLC1
//--------------------------------

CALL FB670, DB 809;

END_FUNCTION


// <SPLIT>CM_INSTANCE_FIC101.awl</SPLIT>


// ___FIC101

// CM Instance DB
// DB811 = FIC101
// FB670 = BST_PIDAIN_400
DATA_BLOCK DB811 FB670
BEGIN
END_DATA_BLOCK

DATA_BLOCK  DB812
// tagstruct_name = PID_interface
STRUCT
	Operator_Setpoint { S7_m_c := 'true' } : REAL;
	Set_SP { S7_m_c := 'true' } : BOOL;
	Output_Value { S7_m_c := 'true' } : REAL;
	Set_Output { S7_m_c := 'true' } : BOOL;
END_STRUCT
BEGIN
END_DATA_BLOCK

FUNCTION "FIC101_FC" : VOID
TITLE =FIC101_FC
// FIC101_FC

AUTHOR :
FAMILY : 'cminst'
NAME : namehead
VERSION : 0.1

BEGIN
NETWORK
TITLE = Change PID Setpoints
//--------------------------------
// The phase FBs write on the operator setpoints of the PID-controller
// To avoid that the setpoints are always overwritten (and blocking operator control)
// we use pulses generated by the phase to set the setpoints only at specific moments
// i_fOCmdSP (setpoint)
// i_fOCmdMANOP (output)
//--------------------------------

// Write the Operator_Setpoint
A	DB812.Set_SP;
JCN J001;

	L DB812.Operator_Setpoint;
	T DB811.i_fOCmdSP;

J001: NOP 0;


// Write the Output_Value
A	DB812.Set_Output;
JCN J002;

	L DB812.Output_Value;
	T DB811.i_fOCmdMANOP;

J002: NOP 0;

NETWORK
TITLE = Main
//--------------------------------
// PLC1
//--------------------------------

CALL FB670, DB 811;

END_FUNCTION



// <SPLIT>EM_INSTANCE_EM_Instance_1.awl</SPLIT>


// ___EM_Instance_1

// EM Instance DB
// EM_Instance_1
// DB718 = EM_Instance_1
// FB702 = EM_I_OUT
DATA_BLOCK DB718 FB702
BEGIN
END_DATA_BLOCK

FUNCTION "EM_Instance_1_FC" : VOID
TITLE =EM_Instance_1_FC
// EM_Instance_1_FC

AUTHOR :
FAMILY : 'eminst'
NAME : namehead
VERSION : 0.1

BEGIN

NETWORK
TITLE = Main
//--------------------------------
//
//--------------------------------

CALL EM_I_OUT, DB 718(
	em_id := 26,
	Pump_RUN := "M100".QNOFF2,
	PIC01_PV := "LIC001".PV,
	LT01_PV := "LT001".QfVal,
	BV_Bottom_OPN := "MV001".QOPEN,
	BV_Bottom_CLS := "MV001".QCLOSE,
	BV_Tran_M04_OPN := "MV003".QOPEN,
	BV_Tran_M04_CLS := "MV003".QCLOSE,
	Pump_ON := "M100".L_ON,
	PIC01_SP := "LIC001".HMI_SP_INT,
	PIC01_AUT := "LIC001".L_AUT,
	PIC01_VAL_OUT := "LIC001".HMI_MAN,
	PIC01_SET_SP := "LIC001".Set_SP,
	PIC01_SET_OUT := "LIC001".Set_Output,
	BV_Bottom_CMD := "MV001".AUT_OP,
	BV_Tran_M04_CMD := "MV003".AUT_OP
)



END_FUNCTION


// <SPLIT>EM_INSTANCE_EM_Instance_2.awl</SPLIT>


// ___EM_Instance_2

// EM Instance DB
// EM_Instance_2
// DB719 = EM_Instance_2
// FB702 = EM_I_OUT
DATA_BLOCK DB719 FB702
BEGIN
END_DATA_BLOCK

FUNCTION "EM_Instance_2_FC" : VOID
TITLE =EM_Instance_2_FC
// EM_Instance_2_FC

AUTHOR :
FAMILY : 'eminst'
NAME : namehead
VERSION : 0.1

BEGIN

NETWORK
TITLE = Main
//--------------------------------
//
//--------------------------------

CALL EM_I_OUT, DB 719(
	em_id := 27,
	Pump_RUN := "M101".QNOFF2,
	PIC01_PV := "LIC002".PV,
	LT01_PV := "LT002".QfVal,
	BV_Bottom_OPN := "MV002".QOPEN,
	BV_Bottom_CLS := "MV002".QCLOSE,
	BV_Tran_M04_OPN := "MV003".QOPEN,
	BV_Tran_M04_CLS := "MV003".QCLOSE,
	Pump_ON := "M101".L_ON,
	PIC01_SP := "LIC002".HMI_SP_INT,
	PIC01_AUT := "LIC002".L_AUT,
	PIC01_VAL_OUT := "LIC002".HMI_MAN,
	PIC01_SET_SP := "LIC002".Set_SP,
	PIC01_SET_OUT := "LIC002".Set_Output,
	BV_Bottom_CMD := "MV002".AUT_OP,
	BV_Tran_M04_CMD := "MV003".AUT_OP
)



END_FUNCTION


// <SPLIT>EM_INSTANCE_EM_Instance_3.awl</SPLIT>


// ___EM_Instance_3

// EM Instance DB
// EM_Instance_3
// DB720 = EM_Instance_3
// FB702 = EM_I_OUT
DATA_BLOCK DB720 FB702
BEGIN
END_DATA_BLOCK

FUNCTION "EM_Instance_3_FC" : VOID
TITLE =EM_Instance_3_FC
// EM_Instance_3_FC

AUTHOR :
FAMILY : 'eminst'
NAME : namehead
VERSION : 0.1

BEGIN

NETWORK
TITLE = Main
//--------------------------------
//
//--------------------------------

CALL EM_I_OUT, DB 720(
	em_id := 28,
	Pump_RUN := "M102".QNOFF2,
	PIC01_PV := "LIC003".PV,
	LT01_PV := "LT003".QfVal,
	BV_Bottom_OPN := "MV003".QOPEN,
	BV_Bottom_CLS := "MV003".QCLOSE,
	BV_Tran_M04_OPN := "MV003".QOPEN,
	BV_Tran_M04_CLS := "MV003".QCLOSE,
	Pump_ON := "M102".L_ON,
	PIC01_SP := "LIC003".HMI_SP_INT,
	PIC01_AUT := "LIC003".L_AUT,
	PIC01_VAL_OUT := "LIC003".HMI_MAN,
	PIC01_SET_SP := "LIC003".Set_SP,
	PIC01_SET_OUT := "LIC003".Set_Output,
	BV_Bottom_CMD := "MV003".AUT_OP,
	BV_Tran_M04_CMD := "MV003".AUT_OP
)



END_FUNCTION


// <SPLIT>EM_INSTANCE_EM_Instance_4.awl</SPLIT>


// ___EM_Instance_4

// EM Instance DB
// EM_Instance_4
// DB721 = EM_Instance_4
// FB702 = EM_I_OUT
DATA_BLOCK DB721 FB702
BEGIN
END_DATA_BLOCK

FUNCTION "EM_Instance_4_FC" : VOID
TITLE =EM_Instance_4_FC
// EM_Instance_4_FC

AUTHOR :
FAMILY : 'eminst'
NAME : namehead
VERSION : 0.1

BEGIN

NETWORK
TITLE = Main
//--------------------------------
//
//--------------------------------

CALL EM_I_OUT, DB 721(
	em_id := 29,
	Pump_RUN := "M103".QNOFF2,
	PIC01_PV := "LIC004".PV,
	LT01_PV := "LT004".QfVal,
	BV_Bottom_OPN := "MV004".QOPEN,
	BV_Bottom_CLS := "MV004".QCLOSE,
	BV_Tran_M04_OPN := "MV003".QOPEN,
	BV_Tran_M04_CLS := "MV003".QCLOSE,
	Pump_ON := "M103".L_ON,
	PIC01_SP := "LIC004".HMI_SP_INT,
	PIC01_AUT := "LIC004".L_AUT,
	PIC01_VAL_OUT := "LIC004".HMI_MAN,
	PIC01_SET_SP := "LIC004".Set_SP,
	PIC01_SET_OUT := "LIC004".Set_Output,
	BV_Bottom_CMD := "MV004".AUT_OP,
	BV_Tran_M04_CMD := "MV003".AUT_OP
)



END_FUNCTION


// <SPLIT>EM_INSTANCE_EM_Instance_5.awl</SPLIT>


// ___EM_Instance_5

// EM Instance DB
// EM_Instance_5
// DB722 = EM_Instance_5
// FB702 = EM_I_OUT
DATA_BLOCK DB722 FB702
BEGIN
END_DATA_BLOCK

FUNCTION "EM_Instance_5_FC" : VOID
TITLE =EM_Instance_5_FC
// EM_Instance_5_FC

AUTHOR :
FAMILY : 'eminst'
NAME : namehead
VERSION : 0.1

BEGIN

NETWORK
TITLE = Main
//--------------------------------
//
//--------------------------------

CALL EM_I_OUT, DB 722(
	em_id := 30,
	Pump_RUN := "M104".QNOFF2,
	PIC01_PV := "LIC005".PV,
	LT01_PV := "LT005".QfVal,
	BV_Bottom_OPN := "MV005".QOPEN,
	BV_Bottom_CLS := "MV005".QCLOSE,
	BV_Tran_M04_OPN := "MV003".QOPEN,
	BV_Tran_M04_CLS := "MV003".QCLOSE,
	Pump_ON := "M104".L_ON,
	PIC01_SP := "LIC005".HMI_SP_INT,
	PIC01_AUT := "LIC005".L_AUT,
	PIC01_VAL_OUT := "LIC005".HMI_MAN,
	PIC01_SET_SP := "LIC005".Set_SP,
	PIC01_SET_OUT := "LIC005".Set_Output,
	BV_Bottom_CMD := "MV005".AUT_OP,
	BV_Tran_M04_CMD := "MV003".AUT_OP
)



END_FUNCTION


// <SPLIT>EM_INSTANCE_EM_Instance_6.awl</SPLIT>


// ___EM_Instance_6

// EM Instance DB
// EM_Instance_6
// DB723 = EM_Instance_6
// FB702 = EM_I_OUT
DATA_BLOCK DB723 FB702
BEGIN
END_DATA_BLOCK

FUNCTION "EM_Instance_6_FC" : VOID
TITLE =EM_Instance_6_FC
// EM_Instance_6_FC

AUTHOR :
FAMILY : 'eminst'
NAME : namehead
VERSION : 0.1

BEGIN

NETWORK
TITLE = Main
//--------------------------------
//
//--------------------------------

CALL EM_I_OUT, DB 723(
	em_id := 31,
	Pump_RUN := "M105".QNOFF2,
	PIC01_PV := "LIC006".PV,
	LT01_PV := "LT006".QfVal,
	BV_Bottom_OPN := "MV006".QOPEN,
	BV_Bottom_CLS := "MV006".QCLOSE,
	BV_Tran_M04_OPN := "MV003".QOPEN,
	BV_Tran_M04_CLS := "MV003".QCLOSE,
	Pump_ON := "M105".L_ON,
	PIC01_SP := "LIC006".HMI_SP_INT,
	PIC01_AUT := "LIC006".L_AUT,
	PIC01_VAL_OUT := "LIC006".HMI_MAN,
	PIC01_SET_SP := "LIC006".Set_SP,
	PIC01_SET_OUT := "LIC006".Set_Output,
	BV_Bottom_CMD := "MV006".AUT_OP,
	BV_Tran_M04_CMD := "MV003".AUT_OP
)



END_FUNCTION


// <SPLIT>EM_INSTANCE_EM_Instance_7.awl</SPLIT>


// ___EM_Instance_7

// EM Instance DB
// EM_Instance_7
// DB724 = EM_Instance_7
// FB702 = EM_I_OUT
DATA_BLOCK DB724 FB702
BEGIN
END_DATA_BLOCK

FUNCTION "EM_Instance_7_FC" : VOID
TITLE =EM_Instance_7_FC
// EM_Instance_7_FC

AUTHOR :
FAMILY : 'eminst'
NAME : namehead
VERSION : 0.1

BEGIN

NETWORK
TITLE = Main
//--------------------------------
//
//--------------------------------

CALL EM_I_OUT, DB 724(
	em_id := 32,
	Pump_RUN := "M106".QNOFF2,
	PIC01_PV := "FIC100".PV,
	LT01_PV := "LT007".QfVal,
	BV_Bottom_OPN := "MV007".QOPEN,
	BV_Bottom_CLS := "MV007".QCLOSE,
	BV_Tran_M04_OPN := "MV003".QOPEN,
	BV_Tran_M04_CLS := "MV003".QCLOSE,
	Pump_ON := "M106".L_ON,
	PIC01_SP := "FIC100".HMI_SP_INT,
	PIC01_AUT := "FIC100".L_AUT,
	PIC01_VAL_OUT := "FIC100".HMI_MAN,
	PIC01_SET_SP := "FIC100".Set_SP,
	PIC01_SET_OUT := "FIC100".Set_Output,
	BV_Bottom_CMD := "MV007".AUT_OP,
	BV_Tran_M04_CMD := "MV003".AUT_OP
)



END_FUNCTION


// <SPLIT>EM_INSTANCE_EM_Instance_8.awl</SPLIT>


// ___EM_Instance_8

// EM Instance DB
// EM_Instance_8
// DB725 = EM_Instance_8
// FB702 = EM_I_OUT
DATA_BLOCK DB725 FB702
BEGIN
END_DATA_BLOCK

FUNCTION "EM_Instance_8_FC" : VOID
TITLE =EM_Instance_8_FC
// EM_Instance_8_FC

AUTHOR :
FAMILY : 'eminst'
NAME : namehead
VERSION : 0.1

BEGIN

NETWORK
TITLE = Main
//--------------------------------
//
//--------------------------------

CALL EM_I_OUT, DB 725(
	em_id := 33,
	Pump_RUN := "M106".QNOFF2,
	PIC01_PV := "FIC101".PV,
	LT01_PV := "LT100".QfVal,
	BV_Bottom_OPN := "MV007".QOPEN,
	BV_Bottom_CLS := "MV007".QCLOSE,
	BV_Tran_M04_OPN := "MV003".QOPEN,
	BV_Tran_M04_CLS := "MV003".QCLOSE,
	Pump_ON := "M106".L_ON,
	PIC01_SP := "FIC101".HMI_SP_INT,
	PIC01_AUT := "FIC101".L_AUT,
	PIC01_VAL_OUT := "FIC101".HMI_MAN,
	PIC01_SET_SP := "FIC101".Set_SP,
	PIC01_SET_OUT := "FIC101".Set_Output,
	BV_Bottom_CMD := "MV007".AUT_OP,
	BV_Tran_M04_CMD := "MV003".AUT_OP
)



END_FUNCTION


// <SPLIT>EM_INSTANCE_EM_Instance_9.awl</SPLIT>


